C07289=1044.179,214.469,399.618,171.280,39.054,157.394
C07290=1044.186,214.718,399.591,171.283,39.057,157.395
C07291=1044.193,214.967,399.564,171.286,39.059,157.395
C07292=1044.198,215.215,399.538,171.287,39.062,157.396
C07293=1044.206,215.464,399.511,171.290,39.064,157.396
C07294=1044.212,215.712,399.483,171.291,39.067,157.397
C07295=1044.219,215.960,399.457,171.294,39.069,157.397
C07296=1044.225,216.209,399.430,171.296,39.072,157.398
C07297=1044.232,216.458,399.403,171.298,39.074,157.399
C07298=1044.238,216.706,399.377,171.300,39.077,157.399
C07299=1044.245,216.955,399.350,171.303,39.079,157.400
C07300=1044.251,217.202,399.323,171.306,39.082,157.400
C07301=1044.258,217.451,399.296,171.307,39.084,157.401
C07302=1044.265,217.700,399.268,171.310,39.087,157.402
C07303=1044.272,217.948,399.242,171.312,39.089,157.402
C07304=1044.277,218.197,399.215,171.314,39.091,157.403
C07305=1044.285,218.445,399.188,171.316,39.094,157.403
C07306=1044.291,218.694,399.161,171.319,39.096,157.404
C07307=1044.298,218.941,399.134,171.320,39.099,157.404
C07308=1044.304,219.190,399.107,171.323,39.101,157.405
C07309=1044.311,219.439,399.079,171.325,39.103,157.406
C07310=1044.318,219.688,399.053,171.328,39.106,157.406
C07311=1044.324,219.936,399.026,171.329,39.109,157.407
C07312=1044.331,220.184,398.999,171.332,39.111,157.407
C07313=1044.338,220.475,398.967,171.335,39.114,157.408
C07314=1044.346,220.766,398.935,171.337,39.117,157.409
C07315=1044.353,221.056,398.903,171.340,39.120,157.409
C07316=1044.362,221.347,398.871,171.343,39.123,157.410
C07317=1044.367,221.596,398.845,171.345,39.125,157.411
C07318=1044.374,221.844,398.817,171.347,39.128,157.411
C07319=1044.381,222.093,398.790,171.349,39.130,157.412
C07320=1044.387,222.341,398.763,171.352,39.133,157.412
C07321=1044.394,222.589,398.735,171.354,39.135,157.413
C07322=1044.400,222.838,398.708,171.356,39.138,157.414
C07323=1044.407,223.087,398.681,171.358,39.140,157.414
C07324=1044.413,223.334,398.653,171.361,39.142,157.415
C07325=1044.420,223.583,398.626,171.364,39.145,157.415
C07326=1044.427,223.831,398.599,171.365,39.148,157.416
C07327=1044.434,224.080,398.571,171.368,39.150,157.417
C07328=1044.439,224.328,398.545,171.370,39.152,157.417
C07329=1044.446,224.577,398.517,171.373,39.155,157.418
C07330=1044.453,224.825,398.489,171.374,39.158,157.418
C07331=1044.459,225.074,398.461,171.377,39.160,157.419
C07332=1044.466,225.323,398.434,171.379,39.162,157.420
C07333=1044.472,225.570,398.407,171.382,39.164,157.420
C07334=1044.479,225.819,398.380,171.385,39.167,157.421
C07335=1044.486,226.067,398.352,171.386,39.170,157.421
C07336=1044.492,226.316,398.325,171.389,39.172,157.422
C07337=1044.499,226.564,398.297,171.391,39.174,157.422
C07338=1044.506,226.813,398.270,171.394,39.177,157.423
C07339=1044.512,227.061,398.242,171.396,39.179,157.424
C07340=1044.519,227.309,398.215,171.398,39.182,157.424
C07341=1044.525,227.558,398.188,171.400,39.184,157.425
C07342=1044.532,227.807,398.160,171.403,39.186,157.425
C07343=1044.539,228.055,398.133,171.405,39.189,157.426
C07344=1044.546,228.303,398.105,171.408,39.192,157.427
C07345=1044.552,228.552,398.077,171.410,39.194,157.427
C07346=1044.559,228.800,398.050,171.412,39.196,157.428
C07347=1044.565,229.048,398.022,171.415,39.199,157.428
C07348=1044.572,229.296,397.994,171.417,39.201,157.429
C07349=1044.578,229.545,397.966,171.420,39.204,157.429
C07350=1044.584,229.793,397.938,171.421,39.206,157.430
C07351=1044.591,230.042,397.911,171.424,39.208,157.431
C07352=1044.598,230.290,397.883,171.427,39.211,157.431
C07353=1044.604,230.539,397.855,171.429,39.214,157.432
C07354=1044.611,230.786,397.828,171.432,39.216,157.432
C07355=1044.617,231.035,397.800,171.434,39.218,157.433
C07356=1044.624,231.283,397.772,171.436,39.221,157.434
C07357=1044.631,231.532,397.745,171.438,39.223,157.434
C07358=1044.637,231.781,397.716,171.441,39.226,157.435
C07359=1044.643,232.029,397.689,171.443,39.228,157.435
C07360=1044.650,232.277,397.661,171.446,39.231,157.436
C07361=1044.657,232.526,397.633,171.449,39.233,157.437
C07362=1044.663,232.774,397.605,171.451,39.236,157.437
C07363=1044.669,233.023,397.577,171.453,39.238,157.438
C07364=1044.675,233.271,397.550,171.455,39.241,157.438
C07365=1044.682,233.519,397.521,171.458,39.243,157.439
C07366=1044.689,233.767,397.494,171.461,39.246,157.440
C07367=1044.695,234.016,397.465,171.463,39.248,157.440
C07368=1044.702,234.264,397.438,171.466,39.251,157.441
C07369=1044.709,234.547,397.405,171.468,39.253,157.441
C07370=1044.717,234.831,397.373,171.471,39.256,157.442
C07371=1044.724,235.114,397.342,171.474,39.259,157.443
C07372=1044.731,235.397,397.309,171.476,39.262,157.444
C07373=1044.738,235.646,397.282,171.479,39.264,157.444
C07374=1044.745,235.894,397.254,171.481,39.267,157.445
C07375=1044.751,236.142,397.225,171.484,39.269,157.445
C07376=1044.758,236.391,397.197,171.487,39.272,157.446
C07377=1044.764,236.639,397.169,171.489,39.274,157.447
C07378=1044.771,236.887,397.142,171.492,39.276,157.447
C07379=1044.777,237.136,397.113,171.494,39.279,157.448
C07380=1044.784,237.384,397.085,171.497,39.282,157.448
C07381=1044.790,237.632,397.057,171.498,39.284,157.449
C07382=1044.797,237.881,397.028,171.501,39.286,157.449
C07383=1044.803,238.129,397.000,171.504,39.289,157.450
C07384=1044.810,238.377,396.972,171.506,39.291,157.451
C07385=1044.816,238.626,396.944,171.509,39.294,157.451
C07386=1044.823,238.874,396.916,171.511,39.296,157.452
C07387=1044.830,239.122,396.887,171.514,39.299,157.453
C07388=1044.837,239.371,396.859,171.516,39.301,157.453
C07389=1044.844,239.619,396.830,171.519,39.303,157.454
C07390=1044.850,239.868,396.803,171.521,39.306,157.454
C07391=1044.856,240.116,396.774,171.524,39.309,157.455
C07392=1044.863,240.364,396.746,171.527,39.311,157.455
C07393=1044.870,240.613,396.718,171.529,39.313,157.456
C07394=1044.876,240.861,396.689,171.532,39.315,157.457
C07395=1044.883,241.109,396.661,171.534,39.318,157.457
C07396=1044.889,241.357,396.632,171.537,39.321,157.458
C07397=1044.896,241.606,396.605,171.540,39.323,157.458
C07398=1044.902,241.854,396.575,171.542,39.326,157.459
C07399=1044.909,242.102,396.547,171.545,39.328,157.460
C07400=1044.915,242.350,396.519,171.547,39.330,157.460
C07401=1044.922,242.599,396.489,171.550,39.333,157.461
C07402=1044.929,242.847,396.461,171.553,39.335,157.462
C07403=1044.935,243.096,396.433,171.554,39.338,157.462
C07404=1044.942,243.344,396.404,171.557,39.341,157.463
C07405=1044.948,243.592,396.376,171.559,39.343,157.463
C07406=1044.954,243.841,396.347,171.562,39.345,157.464
C07407=1044.961,244.088,396.318,171.564,39.348,157.465
C07408=1044.967,244.336,396.289,171.567,39.350,157.465
C07409=1044.974,244.585,396.262,171.570,39.353,157.466
C07410=1044.981,244.834,396.232,171.572,39.355,157.466
C07411=1044.987,245.082,396.203,171.575,39.358,157.467
C07412=1044.994,245.330,396.175,171.577,39.360,157.468
C07413=1045.000,245.578,396.146,171.580,39.363,157.468
C07414=1045.006,245.827,396.117,171.583,39.365,157.469
C07415=1045.012,246.075,396.088,171.585,39.368,157.470
C07416=1045.019,246.323,396.060,171.588,39.370,157.470
C07417=1045.026,246.571,396.031,171.590,39.373,157.471
C07418=1045.032,246.820,396.002,171.593,39.375,157.471
C07419=1045.038,247.068,395.973,171.596,39.378,157.472
C07420=1045.045,247.316,395.944,171.598,39.381,157.473
C07421=1045.051,247.565,395.915,171.601,39.383,157.473
C07422=1045.057,247.813,395.886,171.603,39.386,157.474
C07423=1045.064,248.060,395.857,171.606,39.388,157.474
C07424=1045.070,248.309,395.828,171.610,39.390,157.475
C07425=1045.077,248.587,395.796,171.612,39.393,157.476
C07426=1045.085,248.864,395.764,171.615,39.396,157.476
C07427=1045.092,249.141,395.731,171.618,39.399,157.477
C07428=1045.099,249.419,395.698,171.621,39.402,157.478
C07429=1045.106,249.667,395.670,171.624,39.405,157.479
C07430=1045.112,249.915,395.641,171.627,39.407,157.479
C07431=1045.119,250.164,395.611,171.629,39.409,157.480
C07432=1045.125,250.412,395.582,171.632,39.412,157.480
C07433=1045.131,250.660,395.553,171.634,39.414,157.481
C07434=1045.137,250.908,395.524,171.637,39.417,157.482
C07435=1045.144,251.157,395.495,171.640,39.419,157.482
C07436=1045.151,251.405,395.466,171.642,39.422,157.483
C07437=1045.157,251.653,395.437,171.645,39.424,157.484
C07438=1045.164,251.900,395.408,171.647,39.427,157.484
C07439=1045.171,252.149,395.378,171.650,39.430,157.485
C07440=1045.177,252.397,395.349,171.654,39.432,157.485
C07441=1045.183,252.646,395.320,171.656,39.434,157.486
C07442=1045.190,252.894,395.291,171.659,39.437,157.487
C07443=1045.197,253.143,395.262,171.661,39.439,157.487
C07444=1045.203,253.391,395.233,171.664,39.442,157.488
C07445=1045.209,253.639,395.204,171.667,39.444,157.488
C07446=1045.216,253.887,395.174,171.669,39.447,157.489
C07447=1045.222,254.135,395.145,171.672,39.449,157.490
C07448=1045.229,254.383,395.115,171.674,39.452,157.490
C07449=1045.236,254.632,395.087,171.678,39.454,157.491
C07450=1045.243,254.879,395.057,171.681,39.457,157.492
C07451=1045.249,255.127,395.028,171.683,39.459,157.492
C07452=1045.256,255.376,394.998,171.686,39.462,157.493
C07453=1045.262,255.624,394.969,171.688,39.464,157.493
C07454=1045.269,255.872,394.940,171.691,39.466,157.494
C07455=1045.276,256.121,394.910,171.694,39.469,157.495
C07456=1045.282,256.369,394.881,171.697,39.471,157.495
C07457=1045.289,256.618,394.852,171.700,39.474,157.496
C07458=1045.295,256.865,394.822,171.702,39.477,157.497
C07459=1045.302,257.113,394.793,171.705,39.479,157.497
C07460=1045.308,257.362,394.764,171.708,39.482,157.498
C07461=1045.315,257.610,394.734,171.710,39.484,157.498
C07462=1045.322,257.859,394.704,171.714,39.486,157.499
C07463=1045.329,258.106,394.675,171.717,39.489,157.500
C07464=1045.335,258.354,394.646,171.719,39.491,157.500
C07465=1045.342,258.603,394.617,171.722,39.494,157.501
C07466=1045.349,258.850,394.587,171.724,39.496,157.502
C07467=1045.356,259.099,394.558,171.728,39.498,157.502
C07468=1045.362,259.347,394.528,171.731,39.501,157.503
C07469=1045.369,259.595,394.499,171.733,39.504,157.503
C07470=1045.376,259.843,394.469,171.736,39.506,157.504
C07471=1045.382,260.092,394.439,171.738,39.509,157.505
C07472=1045.389,260.339,394.410,171.742,39.511,157.505
C07473=1045.396,260.588,394.380,171.745,39.513,157.506
C07474=1045.402,260.836,394.350,171.747,39.516,157.507
C07475=1045.409,261.084,394.321,171.750,39.518,157.507
C07476=1045.416,261.332,394.291,171.754,39.521,157.508
C07477=1045.423,261.581,394.262,171.756,39.523,157.508
C07478=1045.429,261.828,394.232,171.759,39.525,157.509
C07479=1045.436,262.077,394.203,171.761,39.528,157.510
C07480=1045.443,262.325,394.173,171.765,39.530,157.510
C07481=1045.450,262.600,394.140,171.768,39.533,157.511
C07482=1045.457,262.876,394.106,171.771,39.536,157.512
C07483=1045.465,263.153,394.074,171.774,39.539,157.513
C07484=1045.472,263.429,394.040,171.778,39.542,157.513
C07485=1045.479,263.677,394.010,171.780,39.545,157.514
C07486=1045.485,263.925,393.980,171.783,39.547,157.515
C07487=1045.492,264.173,393.950,171.786,39.550,157.515
C07488=1045.498,264.421,393.921,171.788,39.552,157.516
C07489=1045.505,264.670,393.890,171.792,39.555,157.517
C07490=1045.511,264.917,393.860,171.794,39.557,157.517
C07491=1045.518,265.165,393.830,171.797,39.560,157.518
C07492=1045.524,265.413,393.800,171.801,39.563,157.519
C07493=1045.531,265.662,393.770,171.803,39.565,157.519
C07494=1045.537,265.910,393.741,171.806,39.568,157.520
C07495=1045.544,266.158,393.710,171.809,39.570,157.520
C07496=1045.551,266.406,393.680,171.812,39.573,157.521
C07497=1045.558,266.654,393.650,171.815,39.575,157.522
C07498=1045.564,266.902,393.619,171.818,39.578,157.522
C07499=1045.571,267.150,393.589,171.820,39.580,157.523
C07500=1045.578,267.398,393.559,171.824,39.583,157.524
C07501=1045.584,267.647,393.529,171.827,39.585,157.524
C07502=1045.591,267.894,393.499,171.829,39.588,157.525
C07503=1045.597,268.143,393.468,171.833,39.591,157.526
C07504=1045.604,268.390,393.438,171.836,39.593,157.526
C07505=1045.610,268.639,393.408,171.838,39.596,157.527
C07506=1045.617,268.886,393.378,171.842,39.598,157.528
C07507=1045.623,269.135,393.347,171.845,39.601,157.528
C07508=1045.630,269.383,393.317,171.847,39.603,157.529
C07509=1045.636,269.631,393.287,171.851,39.606,157.530
C07510=1045.643,269.879,393.257,171.854,39.609,157.530
C07511=1045.650,270.127,393.226,171.856,39.611,157.531
C07512=1045.656,270.375,393.196,171.859,39.614,157.532
C07513=1045.663,270.624,393.165,171.863,39.616,157.532
C07514=1045.670,270.872,393.135,171.865,39.619,157.533
C07515=1045.676,271.119,393.104,171.869,39.621,157.534
C07516=1045.683,271.367,393.074,171.871,39.624,157.534
C07517=1045.689,271.616,393.043,171.874,39.626,157.535
C07518=1045.696,271.863,393.014,171.878,39.629,157.536
C07519=1045.702,272.112,392.983,171.880,39.631,157.536
C07520=1045.709,272.360,392.952,171.883,39.634,157.537
C07521=1045.716,272.607,392.922,171.887,39.637,157.538
C07522=1045.722,272.856,392.891,171.889,39.639,157.538
C07523=1045.729,273.104,392.860,171.892,39.642,157.539
C07524=1045.735,273.351,392.830,171.896,39.645,157.540
C07525=1045.742,273.600,392.799,171.898,39.647,157.540
C07526=1045.748,273.848,392.768,171.901,39.650,157.541
C07527=1045.755,274.095,392.738,171.905,39.653,157.542
C07528=1045.762,274.344,392.707,171.907,39.655,157.542
C07529=1045.768,274.592,392.677,171.911,39.658,157.543
C07530=1045.775,274.840,392.646,171.914,39.660,157.544
C07531=1045.781,275.087,392.615,171.916,39.663,157.544
C07532=1045.788,275.336,392.585,171.920,39.665,157.545
C07533=1045.794,275.584,392.553,171.923,39.668,157.546
C07534=1045.802,275.832,392.523,171.927,39.671,157.547
C07535=1045.808,276.079,392.492,171.929,39.673,157.547
C07536=1045.814,276.328,392.461,171.932,39.676,157.548
C07537=1045.825,276.739,392.410,171.937,39.681,157.549
C07538=1045.832,276.982,392.380,171.941,39.683,157.550
C07539=1045.838,277.225,392.350,171.943,39.686,157.550
C07540=1045.845,277.468,392.319,171.946,39.688,157.551
C07541=1045.851,277.711,392.289,171.950,39.691,157.552
C07542=1045.858,277.954,392.258,171.952,39.693,157.552
C07543=1045.865,278.198,392.228,171.956,39.696,157.553
C07544=1045.871,278.441,392.198,171.959,39.698,157.554
C07545=1045.877,278.690,392.167,171.961,39.701,157.554
C07546=1045.884,278.937,392.136,171.965,39.704,157.555
C07547=1045.891,279.185,392.105,171.968,39.707,157.556
C07548=1045.897,279.433,392.074,171.971,39.709,157.557
C07549=1045.904,279.681,392.043,171.974,39.712,157.557
C07550=1045.911,279.929,392.011,171.978,39.714,157.558
C07551=1045.917,280.177,391.981,171.980,39.717,157.559
C07552=1045.923,280.425,391.950,171.984,39.720,157.559
C07553=1045.930,280.672,391.918,171.987,39.723,157.560
C07554=1045.937,280.920,391.887,171.990,39.726,157.561
C07555=1045.943,281.169,391.856,171.993,39.728,157.561
C07556=1045.950,281.417,391.825,171.996,39.731,157.562
C07557=1045.957,281.665,391.793,172.000,39.733,157.563
C07558=1045.963,281.912,391.762,172.002,39.736,157.564
C07559=1045.969,282.160,391.730,172.006,39.739,157.564
C07560=1045.976,282.408,391.699,172.009,39.742,157.565
C07561=1045.982,282.657,391.668,172.013,39.744,157.566
C07562=1045.989,282.904,391.637,172.015,39.747,157.566
C07563=1045.995,283.152,391.605,172.019,39.749,157.567
C07564=1046.002,283.400,391.574,172.022,39.752,157.568
C07565=1046.009,283.648,391.542,172.025,39.755,157.568
C07566=1046.016,283.896,391.511,172.028,39.758,157.569
C07567=1046.022,284.144,391.479,172.032,39.760,157.570
C07568=1046.029,284.392,391.448,172.035,39.763,157.571
C07569=1046.036,284.640,391.416,172.038,39.766,157.571
C07570=1046.043,284.888,391.385,172.041,39.769,157.572
C07571=1046.049,285.136,391.354,172.045,39.772,157.573
C07572=1046.056,285.383,391.322,172.047,39.774,157.573
C07573=1046.063,285.631,391.291,172.051,39.776,157.574
C07574=1046.069,285.879,391.259,172.055,39.779,157.575
C07575=1046.076,286.127,391.228,172.058,39.782,157.576
C07576=1046.083,286.375,391.196,172.061,39.785,157.576
C07577=1046.090,286.623,391.165,172.064,39.788,157.577
C07578=1046.096,286.871,391.134,172.068,39.790,157.578
C07579=1046.103,287.119,391.102,172.070,39.793,157.579
C07580=1046.110,287.367,391.071,172.074,39.796,157.579
C07581=1046.116,287.615,391.039,172.078,39.799,157.580
C07582=1046.123,287.862,391.007,172.081,39.801,157.581
C07583=1046.130,288.110,390.975,172.084,39.804,157.581
C07584=1046.136,288.358,390.944,172.087,39.807,157.582
C07585=1046.142,288.606,390.912,172.091,39.810,157.583
C07586=1046.149,288.853,390.880,172.094,39.812,157.584
C07587=1046.156,289.101,390.848,172.097,39.815,157.584
C07588=1046.163,289.349,390.817,172.101,39.818,157.585
C07589=1046.169,289.598,390.785,172.104,39.821,157.586
C07590=1046.176,289.845,390.752,172.108,39.823,157.587
C07591=1046.182,290.093,390.721,172.110,39.826,157.587
C07592=1046.189,290.341,390.690,172.114,39.829,157.588
C07593=1046.197,290.633,390.652,172.118,39.832,157.589
C07594=1046.205,290.924,390.613,172.122,39.835,157.590
C07595=1046.212,291.216,390.576,172.126,39.839,157.591
C07596=1046.220,291.509,390.538,172.130,39.842,157.592
C07597=1046.227,291.757,390.506,172.133,39.845,157.592
C07598=1046.234,292.004,390.474,172.136,39.848,157.593
C07599=1046.240,292.252,390.442,172.140,39.850,157.594
C07600=1046.247,292.500,390.410,172.144,39.853,157.595
C07601=1046.254,292.748,390.379,172.146,39.856,157.595
C07602=1046.260,292.995,390.346,172.150,39.859,157.596
C07603=1046.268,293.244,390.314,172.154,39.862,157.597
C07604=1046.275,293.491,390.282,172.157,39.865,157.598
C07605=1046.281,293.739,390.250,172.160,39.867,157.598
C07606=1046.288,293.987,390.218,172.164,39.870,157.599
C07607=1046.294,294.235,390.186,172.167,39.873,157.600
C07608=1046.301,294.482,390.154,172.171,39.876,157.601
C07609=1046.308,294.730,390.121,172.174,39.878,157.601
C07610=1046.314,294.978,390.089,172.177,39.882,157.602
C07611=1046.321,295.226,390.056,172.181,39.884,157.603
C07612=1046.328,295.473,390.024,172.185,39.887,157.604
C07613=1046.334,295.721,389.993,172.187,39.890,157.604
C07614=1046.341,295.969,389.960,172.191,39.893,157.605
C07615=1046.348,296.217,389.927,172.195,39.896,157.606
C07616=1046.354,296.465,389.894,172.198,39.899,157.607
C07617=1046.361,296.712,389.863,172.202,39.901,157.607
C07618=1046.367,296.960,389.830,172.206,39.905,157.608
C07619=1046.373,297.208,389.797,172.208,39.908,157.609
C07620=1046.380,297.456,389.764,172.212,39.910,157.610
C07621=1046.386,297.703,389.731,172.216,39.914,157.611
C07622=1046.393,297.951,389.699,172.219,39.916,157.611
C07623=1046.400,298.198,389.667,172.223,39.920,157.612
C07624=1046.407,298.447,389.633,172.226,39.922,157.613
C07625=1046.413,298.695,389.601,172.229,39.925,157.614
C07626=1046.420,298.942,389.569,172.233,39.928,157.615
C07627=1046.426,299.190,389.537,172.237,39.931,157.615
C07628=1046.433,299.438,389.503,172.241,39.934,157.616
C07629=1046.439,299.686,389.471,172.243,39.937,157.617
C07630=1046.445,299.933,389.438,172.247,39.940,157.618
C07631=1046.452,300.180,389.406,172.251,39.943,157.619
C07632=1046.459,300.429,389.373,172.254,39.946,157.619
C07633=1046.466,300.676,389.339,172.258,39.949,157.620
C07634=1046.472,300.923,389.306,172.261,39.952,157.621
C07635=1046.479,301.172,389.273,172.265,39.955,157.622
C07636=1046.485,301.419,389.241,172.268,39.958,157.623
C07637=1046.492,301.667,389.208,172.272,39.961,157.623
C07638=1046.499,301.915,389.175,172.276,39.964,157.624
C07639=1046.506,302.162,389.143,172.279,39.967,157.625
C07640=1046.512,302.410,389.110,172.282,39.970,157.626
C07641=1046.519,302.658,389.077,172.286,39.973,157.627
C07642=1046.525,302.905,389.043,172.290,39.975,157.627
C07643=1046.532,303.153,389.011,172.294,39.979,157.628
C07644=1046.539,303.401,388.978,172.298,39.981,157.629
C07645=1046.546,303.648,388.945,172.300,39.985,157.630
C07646=1046.553,303.896,388.912,172.304,39.987,157.631
C07647=1046.559,304.144,388.879,172.308,39.991,157.632
C07648=1046.565,304.391,388.846,172.312,39.993,157.632
C07649=1046.575,304.699,388.805,172.316,39.997,157.633
C07650=1046.582,305.008,388.764,172.321,40.001,157.634
C07651=1046.591,305.316,388.723,172.325,40.005,157.635
C07652=1046.600,305.624,388.681,172.330,40.009,157.636
C07653=1046.606,305.872,388.648,172.334,40.011,157.637
C07654=1046.613,306.120,388.615,172.338,40.015,157.638
C07655=1046.620,306.367,388.582,172.341,40.017,157.639
C07656=1046.627,306.615,388.549,172.344,40.021,157.640
C07657=1046.634,306.862,388.516,172.348,40.023,157.640
C07658=1046.641,307.111,388.482,172.352,40.027,157.641
C07659=1046.647,307.358,388.450,172.356,40.029,157.642
C07660=1046.654,307.606,388.416,172.360,40.033,157.643
C07661=1046.661,307.853,388.383,172.364,40.035,157.644
C07662=1046.668,308.101,388.349,172.368,40.039,157.645
C07663=1046.675,308.348,388.317,172.370,40.042,157.646
C07664=1046.682,308.596,388.283,172.374,40.045,157.646
C07665=1046.689,308.844,388.250,172.378,40.048,157.647
C07666=1046.696,309.091,388.217,172.382,40.051,157.648
C07667=1046.703,309.339,388.183,172.386,40.054,157.649
C07668=1046.709,309.587,388.150,172.390,40.057,157.650
C07669=1046.716,309.834,388.116,172.393,40.060,157.650
C07670=1046.723,310.082,388.083,172.397,40.063,157.651
C07671=1046.730,310.330,388.050,172.401,40.066,157.652
C07672=1046.737,310.577,388.016,172.405,40.069,157.653
C07673=1046.744,310.826,387.983,172.409,40.072,157.654
C07674=1046.751,311.072,387.950,172.412,40.075,157.655
C07675=1046.758,311.320,387.916,172.416,40.078,157.656
C07676=1046.766,311.568,387.882,172.420,40.082,157.656
C07677=1046.772,311.815,387.850,172.423,40.084,157.657
C07678=1046.779,312.063,387.816,172.427,40.087,157.658
C07679=1046.786,312.310,387.782,172.431,40.091,157.659
C07680=1046.794,312.558,387.748,172.435,40.093,157.660
C07681=1046.800,312.806,387.715,172.439,40.097,157.661
C07682=1046.806,313.054,387.681,172.443,40.100,157.662
C07683=1046.813,313.301,387.647,172.447,40.103,157.662
C07684=1046.819,313.549,387.613,172.451,40.106,157.663
C07685=1046.827,313.796,387.579,172.455,40.110,157.664
C07686=1046.834,314.044,387.546,172.459,40.113,157.665
C07687=1046.840,314.291,387.511,172.462,40.116,157.666
C07688=1046.847,314.539,387.478,172.466,40.119,157.667
C07689=1046.854,314.786,387.442,172.470,40.123,157.668
C07690=1046.860,315.033,387.409,172.474,40.126,157.669
C07691=1046.867,315.281,387.375,172.477,40.129,157.670
C07692=1046.874,315.529,387.341,172.481,40.133,157.670
C07693=1046.880,315.776,387.307,172.485,40.136,157.671
C07694=1046.887,316.024,387.273,172.489,40.139,157.672
C07695=1046.893,316.272,387.238,172.493,40.142,157.673
C07696=1046.901,316.520,387.205,172.497,40.146,157.674
C07697=1046.907,316.766,387.170,172.501,40.149,157.675
C07698=1046.914,317.014,387.136,172.505,40.152,157.676
C07699=1046.920,317.262,387.102,172.509,40.155,157.677
C07700=1046.928,317.510,387.068,172.513,40.159,157.678
C07701=1046.934,317.758,387.033,172.516,40.162,157.679
C07702=1046.941,318.004,386.999,172.520,40.165,157.679
C07703=1046.947,318.252,386.965,172.524,40.168,157.680
C07704=1046.955,318.500,386.931,172.528,40.172,157.681
C07705=1046.963,318.812,386.887,172.534,40.176,157.682
C07706=1046.971,319.125,386.844,172.539,40.180,157.684
C07707=1046.980,319.438,386.800,172.544,40.184,157.685
C07708=1046.989,319.751,386.757,172.549,40.188,157.686
C07709=1046.996,319.999,386.723,172.553,40.191,157.687
C07710=1047.003,320.246,386.688,172.557,40.195,157.688
C07711=1047.010,320.494,386.654,172.561,40.198,157.689
C07712=1047.016,320.740,386.619,172.565,40.202,157.690
C07713=1047.023,320.988,386.585,172.569,40.205,157.691
C07714=1047.030,321.235,386.551,172.573,40.208,157.691
C07715=1047.037,321.483,386.516,172.577,40.212,157.692
C07716=1047.044,321.730,386.481,172.581,40.215,157.693
C07717=1047.051,321.978,386.447,172.585,40.218,157.694
C07718=1047.058,322.226,386.412,172.589,40.222,157.695
C07719=1047.065,322.473,386.378,172.593,40.225,157.696
C07720=1047.072,322.721,386.343,172.598,40.228,157.697
C07721=1047.079,322.968,386.309,172.602,40.231,157.698
C07722=1047.086,323.216,386.274,172.606,40.235,157.699
C07723=1047.092,323.463,386.239,172.610,40.238,157.700
C07724=1047.100,323.711,386.205,172.614,40.242,157.701
C07725=1047.106,323.958,386.170,172.618,40.245,157.702
C07726=1047.114,324.206,386.135,172.622,40.248,157.703
C07727=1047.121,324.454,386.101,172.626,40.252,157.704
C07728=1047.128,324.701,386.066,172.631,40.255,157.705
C07729=1047.135,324.948,386.031,172.635,40.258,157.705
C07730=1047.142,325.196,385.997,172.639,40.262,157.707
C07731=1047.149,325.443,385.962,172.643,40.265,157.707
C07732=1047.156,325.691,385.927,172.647,40.269,157.708
C07733=1047.163,325.938,385.892,172.651,40.272,157.709
C07734=1047.170,326.185,385.857,172.656,40.275,157.710
C07735=1047.177,326.434,385.822,172.660,40.279,157.711
C07736=1047.185,326.681,385.788,172.664,40.283,157.712
C07737=1047.192,326.928,385.753,172.668,40.286,157.713
C07738=1047.198,327.175,385.718,172.672,40.289,157.714
C07739=1047.206,327.422,385.683,172.677,40.293,157.715
C07740=1047.213,327.671,385.648,172.681,40.296,157.716
C07741=1047.220,327.918,385.612,172.685,40.300,157.717
C07742=1047.227,328.165,385.578,172.689,40.303,157.718
C07743=1047.234,328.412,385.543,172.693,40.306,157.719
C07744=1047.242,328.660,385.508,172.698,40.310,157.720
C07745=1047.249,328.907,385.473,172.702,40.313,157.721
C07746=1047.256,329.155,385.438,172.706,40.317,157.722
C07747=1047.263,329.402,385.403,172.710,40.320,157.723
C07748=1047.271,329.650,385.368,172.715,40.324,157.724
C07749=1047.277,329.897,385.332,172.719,40.327,157.725
C07750=1047.284,330.145,385.297,172.723,40.331,157.726
C07751=1047.291,330.392,385.262,172.727,40.335,157.727
C07752=1047.299,330.639,385.226,172.732,40.338,157.728
C07753=1047.305,330.887,385.191,172.736,40.341,157.729
C07754=1047.312,331.134,385.156,172.740,40.345,157.730
C07755=1047.319,331.382,385.121,172.744,40.349,157.731
C07756=1047.327,331.629,385.084,172.748,40.352,157.732
C07757=1047.333,331.876,385.049,172.753,40.356,157.733
C07758=1047.339,332.124,385.013,172.758,40.360,157.734
C07759=1047.347,332.372,384.977,172.762,40.363,157.735
C07760=1047.354,332.619,384.942,172.767,40.367,157.736
C07761=1047.362,332.926,384.898,172.772,40.371,157.737
C07762=1047.371,333.235,384.854,172.777,40.376,157.739
C07763=1047.381,333.542,384.809,172.783,40.381,157.740
C07764=1047.389,333.850,384.765,172.788,40.385,157.741
C07765=1047.396,334.098,384.730,172.792,40.389,157.742
C07766=1047.403,334.345,384.694,172.797,40.392,157.743
C07767=1047.410,334.592,384.659,172.802,40.396,157.744
C07768=1047.418,334.839,384.622,172.805,40.399,157.745
C07769=1047.425,335.087,384.587,172.811,40.403,157.746
C07770=1047.432,335.334,384.551,172.815,40.407,157.747
C07771=1047.439,335.581,384.515,172.819,40.411,157.748
C07772=1047.447,335.829,384.480,172.824,40.414,157.750
C07773=1047.454,336.076,384.444,172.828,40.418,157.751
C07774=1047.460,336.323,384.407,172.832,40.422,157.752
C07775=1047.468,336.571,384.372,172.837,40.425,157.753
C07776=1047.475,336.818,384.336,172.842,40.429,157.754
C07777=1047.482,337.065,384.299,172.846,40.433,157.755
C07778=1047.488,337.313,384.264,172.851,40.437,157.756
C07779=1047.496,337.560,384.228,172.855,40.440,157.757
C07780=1047.502,337.807,384.191,172.859,40.444,157.758
C07781=1047.510,338.055,384.155,172.864,40.448,157.759
C07782=1047.517,338.301,384.119,172.868,40.452,157.760
C07783=1047.524,338.549,384.083,172.873,40.456,157.761
C07784=1047.531,338.797,384.047,172.878,40.460,157.763
C07785=1047.538,339.044,384.011,172.882,40.463,157.764
C07786=1047.546,339.291,383.975,172.887,40.467,157.765
C07787=1047.552,339.539,383.939,172.891,40.471,157.766
C07788=1047.560,339.785,383.903,172.896,40.475,157.767
C07789=1047.567,340.033,383.867,172.901,40.479,157.768
C07790=1047.574,340.280,383.830,172.905,40.483,157.769
C07791=1047.581,340.527,383.794,172.910,40.486,157.770
C07792=1047.589,340.775,383.758,172.914,40.490,157.771
C07793=1047.596,341.022,383.721,172.919,40.494,157.772
C07794=1047.603,341.269,383.685,172.924,40.498,157.773
C07795=1047.610,341.517,383.648,172.929,40.502,157.775
C07796=1047.617,341.764,383.612,172.933,40.505,157.776
C07797=1047.625,342.010,383.575,172.938,40.509,157.777
C07798=1047.632,342.258,383.539,172.942,40.513,157.778
C07799=1047.640,342.506,383.502,172.946,40.517,157.779
C07800=1047.646,342.753,383.466,172.952,40.521,157.780
C07801=1047.654,343.000,383.430,172.956,40.525,157.781
C07802=1047.661,343.247,383.392,172.961,40.529,157.782
C07803=1047.668,343.494,383.356,172.965,40.533,157.784
C07804=1047.675,343.742,383.319,172.970,40.537,157.785
C07805=1047.683,343.989,383.283,172.975,40.541,157.786
C07806=1047.689,344.236,383.246,172.980,40.545,157.787
C07807=1047.696,344.483,383.209,172.984,40.549,157.788
C07808=1047.704,344.730,383.172,172.989,40.553,157.789
C07809=1047.711,344.978,383.136,172.994,40.557,157.790
C07810=1047.718,345.224,383.099,172.999,40.561,157.792
C07811=1047.725,345.472,383.062,173.003,40.565,157.793
C07812=1047.733,345.719,383.025,173.009,40.569,157.794
C07813=1047.740,345.967,382.988,173.013,40.573,157.795
C07814=1047.747,346.213,382.951,173.018,40.577,157.796
C07815=1047.754,346.461,382.914,173.023,40.581,157.797
C07816=1047.762,346.708,382.878,173.027,40.585,157.799
C07817=1047.770,347.012,382.832,173.033,40.591,157.800
C07818=1047.780,347.316,382.786,173.040,40.595,157.802
C07819=1047.788,347.619,382.740,173.045,40.601,157.803
C07820=1047.797,347.923,382.696,173.052,40.605,157.804
C07821=1047.804,348.170,382.658,173.056,40.610,157.806
C07822=1047.812,348.417,382.621,173.061,40.614,157.807
C07823=1047.819,348.665,382.585,173.066,40.618,157.808
C07824=1047.826,348.912,382.547,173.071,40.622,157.809
C07825=1047.834,349.159,382.509,173.076,40.626,157.810
C07826=1047.842,349.406,382.473,173.081,40.630,157.812
C07827=1047.848,349.654,382.436,173.086,40.635,157.813
C07828=1047.856,349.901,382.398,173.090,40.638,157.814
C07829=1047.864,350.148,382.361,173.095,40.642,157.815
C07830=1047.871,350.395,382.324,173.101,40.647,157.816
C07831=1047.878,350.642,382.286,173.105,40.651,157.818
C07832=1047.885,350.889,382.249,173.110,40.655,157.819
C07833=1047.893,351.136,382.211,173.116,40.659,157.820
C07834=1047.900,351.383,382.174,173.120,40.664,157.821
C07835=1047.907,351.631,382.136,173.125,40.668,157.823
C07836=1047.914,351.878,382.099,173.131,40.672,157.824
C07837=1047.922,352.125,382.061,173.135,40.676,157.825
C07838=1047.929,352.372,382.024,173.140,40.681,157.826
C07839=1047.936,352.619,381.986,173.146,40.685,157.828
C07840=1047.944,352.865,381.948,173.150,40.690,157.829
C07841=1047.952,353.112,381.911,173.156,40.694,157.830
C07842=1047.959,353.360,381.873,173.161,40.698,157.831
C07843=1047.966,353.607,381.836,173.165,40.702,157.833
C07844=1047.973,353.854,381.798,173.171,40.706,157.834
C07845=1047.981,354.100,381.760,173.176,40.711,157.835
C07846=1047.988,354.348,381.722,173.182,40.715,157.837
C07847=1047.995,354.595,381.685,173.186,40.720,157.838
C07848=1048.003,354.842,381.647,173.191,40.724,157.839
C07849=1048.010,355.088,381.609,173.197,40.728,157.840
C07850=1048.018,355.336,381.571,173.202,40.733,157.842
C07851=1048.026,355.583,381.533,173.206,40.737,157.843
C07852=1048.033,355.830,381.495,173.212,40.741,157.844
C07853=1048.040,356.077,381.458,173.217,40.746,157.846
C07854=1048.048,356.323,381.420,173.223,40.750,157.847
C07855=1048.056,356.571,381.382,173.227,40.754,157.848
C07856=1048.063,356.818,381.344,173.233,40.759,157.849
C07857=1048.070,357.065,381.306,173.238,40.763,157.851
C07858=1048.078,357.311,381.268,173.243,40.768,157.852
C07859=1048.084,357.559,381.230,173.249,40.772,157.853
C07860=1048.093,357.806,381.191,173.253,40.777,157.855
C07861=1048.100,358.053,381.153,173.259,40.781,157.856
C07862=1048.107,358.300,381.115,173.264,40.786,157.857
C07863=1048.115,358.546,381.077,173.270,40.790,157.859
C07864=1048.123,358.793,381.038,173.275,40.795,157.860
C07865=1048.130,359.040,381.000,173.280,40.800,157.861
C07866=1048.137,359.287,380.962,173.285,40.804,157.863
C07867=1048.145,359.535,380.923,173.291,40.809,157.864
C07868=1048.153,359.781,380.885,173.296,40.813,157.865
C07869=1048.160,360.028,380.847,173.302,40.818,157.867
C07870=1048.168,360.275,380.808,173.307,40.822,157.868
C07871=1048.175,360.522,380.770,173.313,40.827,157.869
C07872=1048.183,360.769,380.732,173.317,40.831,157.871
C07873=1048.193,361.078,380.683,173.324,40.837,157.872
C07874=1048.201,361.387,380.635,173.331,40.843,157.874
C07875=1048.211,361.697,380.587,173.338,40.849,157.876
C07876=1048.221,362.007,380.538,173.345,40.855,157.878
C07877=1048.228,362.253,380.500,173.350,40.859,157.879
C07878=1048.236,362.500,380.461,173.356,40.864,157.880
C07879=1048.243,362.747,380.422,173.361,40.868,157.882
C07880=1048.251,362.994,380.384,173.367,40.873,157.883
C07881=1048.259,363.241,380.345,173.372,40.878,157.885
C07882=1048.266,363.488,380.307,173.377,40.883,157.886
C07883=1048.274,363.734,380.267,173.382,40.887,157.887
C07884=1048.281,363.981,380.228,173.388,40.892,157.889
C07885=1048.288,364.229,380.189,173.394,40.897,157.890
C07886=1048.296,364.475,380.151,173.399,40.902,157.892
C07887=1048.304,364.722,380.111,173.405,40.907,157.893
C07888=1048.311,364.969,380.073,173.410,40.912,157.895
C07889=1048.319,365.216,380.034,173.416,40.916,157.896
C07890=1048.327,365.462,379.995,173.421,40.921,157.897
C07891=1048.334,365.709,379.955,173.427,40.926,157.899
C07892=1048.342,365.955,379.916,173.433,40.931,157.900
C07893=1048.349,366.203,379.877,173.438,40.936,157.902
C07894=1048.358,366.449,379.838,173.444,40.940,157.903
C07895=1048.365,366.696,379.799,173.450,40.946,157.905
C07896=1048.373,366.943,379.760,173.455,40.950,157.906
C07897=1048.380,367.190,379.721,173.461,40.955,157.907
C07898=1048.388,367.437,379.681,173.466,40.960,157.909
C07899=1048.396,367.683,379.642,173.472,40.965,157.910
C07900=1048.403,367.930,379.603,173.478,40.970,157.912
C07901=1048.411,368.177,379.564,173.483,40.975,157.913
C07902=1048.419,368.424,379.524,173.489,40.980,157.915
C07903=1048.427,368.670,379.485,173.496,40.985,157.916
C07904=1048.434,368.917,379.445,173.501,40.989,157.918
C07905=1048.442,369.164,379.406,173.507,40.995,157.919
C07906=1048.450,369.410,379.366,173.513,41.000,157.921
C07907=1048.457,369.657,379.327,173.518,41.005,157.922
C07908=1048.466,369.904,379.288,173.524,41.010,157.924
C07909=1048.473,370.151,379.248,173.530,41.014,157.925
C07910=1048.481,370.398,379.208,173.535,41.020,157.927
C07911=1048.489,370.644,379.169,173.541,41.025,157.929
C07912=1048.497,370.890,379.129,173.548,41.029,157.930
C07913=1048.505,371.137,379.090,173.554,41.035,157.932
C07914=1048.513,371.384,379.050,173.559,41.040,157.933
C07915=1048.521,371.631,379.010,173.565,41.045,157.935
C07916=1048.528,371.878,378.970,173.571,41.050,157.936
C07917=1048.535,372.124,378.931,173.576,41.055,157.938
C07918=1048.543,372.371,378.891,173.583,41.060,157.939
C07919=1048.551,372.618,378.851,173.589,41.065,157.941
C07920=1048.560,372.864,378.811,173.595,41.071,157.942
C07921=1048.567,373.111,378.771,173.600,41.076,157.944
C07922=1048.575,373.358,378.731,173.606,41.081,157.946
C07923=1048.582,373.604,378.691,173.612,41.086,157.947
C07924=1048.590,373.850,378.651,173.619,41.091,157.949
C07925=1048.598,374.097,378.611,173.625,41.097,157.950
C07926=1048.606,374.344,378.571,173.630,41.102,157.952
C07927=1048.614,374.590,378.530,173.636,41.108,157.954
C07928=1048.621,374.837,378.490,173.643,41.113,157.955
C07929=1048.632,375.165,378.436,173.650,41.120,157.957
C07930=1048.643,375.494,378.383,173.659,41.127,157.959
C07931=1048.654,375.823,378.330,173.667,41.134,157.962
C07932=1048.664,376.151,378.276,173.675,41.141,157.964
C07933=1048.671,376.398,378.236,173.682,41.147,157.965
C07934=1048.680,376.645,378.195,173.687,41.152,157.967
C07935=1048.688,376.891,378.155,173.693,41.157,157.969
C07936=1048.696,377.138,378.115,173.700,41.163,157.970
C07937=1048.704,377.384,378.074,173.706,41.168,157.972
C07938=1048.712,377.630,378.033,173.712,41.173,157.973
C07939=1048.720,377.877,377.993,173.719,41.179,157.975
C07940=1048.728,378.124,377.953,173.725,41.184,157.977
C07941=1048.736,378.370,377.912,173.731,41.190,157.979
C07942=1048.744,378.616,377.871,173.737,41.195,157.980
C07943=1048.752,378.863,377.830,173.743,41.200,157.982
C07944=1048.760,379.110,377.791,173.749,41.206,157.984
C07945=1048.768,379.356,377.750,173.756,41.211,157.985
C07946=1048.776,379.603,377.709,173.762,41.217,157.987
C07947=1048.785,379.850,377.668,173.769,41.223,157.989
C07948=1048.793,380.096,377.628,173.775,41.228,157.990
C07949=1048.800,380.343,377.586,173.781,41.234,157.992
C07950=1048.808,380.589,377.546,173.788,41.239,157.994
C07951=1048.816,380.834,377.504,173.794,41.245,157.996
C07952=1048.825,381.081,377.463,173.801,41.251,157.997
C07953=1048.832,381.328,377.422,173.807,41.256,157.999
C07954=1048.840,381.574,377.382,173.814,41.262,158.001
C07955=1048.848,381.821,377.341,173.820,41.268,158.003
C07956=1048.857,382.067,377.299,173.826,41.273,158.004
C07957=1048.865,382.314,377.258,173.833,41.279,158.006
C07958=1048.873,382.560,377.217,173.839,41.285,158.008
C07959=1048.881,382.807,377.175,173.846,41.290,158.010
C07960=1048.889,383.053,377.134,173.852,41.296,158.011
C07961=1048.897,383.299,377.094,173.859,41.302,158.013
C07962=1048.906,383.546,377.052,173.865,41.307,158.015
C07963=1048.913,383.792,377.011,173.872,41.314,158.017
C07964=1048.921,384.038,376.970,173.878,41.319,158.018
C07965=1048.930,384.285,376.929,173.885,41.325,158.020
C07966=1048.938,384.531,376.887,173.891,41.331,158.022
C07967=1048.946,384.778,376.846,173.898,41.337,158.024
C07968=1048.954,385.024,376.804,173.905,41.342,158.026
C07969=1048.963,385.270,376.762,173.911,41.348,158.027
C07970=1048.971,385.516,376.721,173.918,41.354,158.029
C07971=1048.979,385.763,376.679,173.924,41.360,158.031
C07972=1048.987,386.009,376.638,173.932,41.366,158.033
C07973=1048.996,386.256,376.597,173.939,41.372,158.035
C07974=1049.004,386.502,376.555,173.945,41.378,158.037
C07975=1049.012,386.748,376.513,173.952,41.384,158.038
C07976=1049.021,386.994,376.472,173.958,41.390,158.040
C07977=1049.029,387.240,376.429,173.965,41.395,158.042
C07978=1049.038,387.487,376.388,173.972,41.402,158.044
C07979=1049.046,387.733,376.347,173.979,41.408,158.046
C07980=1049.054,387.980,376.305,173.986,41.413,158.048
C07981=1049.063,388.226,376.263,173.993,41.419,158.050
C07982=1049.071,388.472,376.221,174.000,41.426,158.052
C07983=1049.080,388.718,376.179,174.006,41.432,158.054
C07984=1049.089,388.965,376.138,174.013,41.437,158.055
C07985=1049.100,389.326,376.076,174.024,41.447,158.058
C07986=1049.113,389.687,376.013,174.034,41.456,158.061
C07987=1049.125,390.048,375.952,174.044,41.465,158.064
C07988=1049.137,390.410,375.890,174.055,41.474,158.067
C07989=1049.146,390.656,375.848,174.061,41.480,158.069
C07990=1049.154,390.902,375.805,174.068,41.486,158.071
C07991=1049.162,391.149,375.763,174.075,41.492,158.073
C07992=1049.171,391.395,375.721,174.083,41.499,158.075
C07993=1049.180,391.641,375.678,174.090,41.505,158.077
C07994=1049.188,391.886,375.636,174.096,41.511,158.078
C07995=1049.196,392.133,375.594,174.104,41.518,158.081
C07996=1049.205,392.379,375.551,174.111,41.524,158.083
C07997=1049.213,392.626,375.509,174.118,41.530,158.084
C07998=1049.222,392.872,375.466,174.126,41.537,158.087
C07999=1049.231,393.118,375.424,174.133,41.543,158.089
C08000=1049.239,393.364,375.381,174.139,41.550,158.091
C08001=1049.248,393.610,375.338,174.147,41.556,158.093
C08002=1049.255,393.856,375.295,174.154,41.562,158.095
C08003=1049.264,394.102,375.253,174.161,41.569,158.097
C08004=1049.273,394.348,375.210,174.169,41.575,158.099
C08005=1049.281,394.594,375.167,174.176,41.582,158.101
C08006=1049.290,394.840,375.124,174.184,41.588,158.103
C08007=1049.298,395.086,375.081,174.191,41.595,158.105
C08008=1049.307,395.332,375.038,174.198,41.601,158.107
C08009=1049.315,395.578,374.995,174.206,41.608,158.109
C08010=1049.325,395.825,374.952,174.213,41.614,158.111
C08011=1049.334,396.071,374.909,174.221,41.621,158.113
C08012=1049.342,396.317,374.866,174.228,41.627,158.115
C08013=1049.351,396.563,374.823,174.236,41.634,158.117
C08014=1049.359,396.809,374.780,174.243,41.641,158.120
C08015=1049.368,397.055,374.737,174.251,41.647,158.122
C08016=1049.376,397.301,374.694,174.258,41.654,158.124
C08017=1049.385,397.547,374.651,174.266,41.661,158.126
C08018=1049.394,397.793,374.607,174.273,41.668,158.128
C08019=1049.403,398.039,374.564,174.281,41.674,158.130
C08020=1049.411,398.285,374.521,174.288,41.681,158.132
C08021=1049.420,398.531,374.477,174.296,41.687,158.135
C08022=1049.428,398.777,374.434,174.303,41.695,158.137
C08023=1049.438,399.023,374.390,174.311,41.701,158.139
C08024=1049.446,399.269,374.347,174.319,41.708,158.141
C08025=1049.455,399.514,374.303,174.326,41.715,158.143
C08026=1049.464,399.762,374.259,174.334,41.722,158.146
C08027=1049.472,400.007,374.216,174.341,41.729,158.148
C08028=1049.481,400.253,374.173,174.349,41.736,158.150
C08029=1049.490,400.499,374.129,174.358,41.742,158.152
C08030=1049.499,400.745,374.086,174.365,41.749,158.154
C08031=1049.508,400.991,374.041,174.373,41.756,158.157
C08032=1049.517,401.237,373.998,174.380,41.763,158.159
C08033=1049.526,401.482,373.954,174.388,41.770,158.161
C08034=1049.534,401.729,373.910,174.397,41.777,158.163
C08035=1049.543,401.975,373.866,174.405,41.784,158.166
C08036=1049.552,402.221,373.822,174.412,41.791,158.168
C08037=1049.561,402.466,373.778,174.420,41.798,158.170
C08038=1049.570,402.713,373.734,174.428,41.806,158.173
C08039=1049.579,402.958,373.690,174.436,41.813,158.175
C08040=1049.588,403.204,373.646,174.444,41.820,158.177
C08041=1049.601,403.585,373.578,174.456,41.831,158.181
C08042=1049.616,403.965,373.509,174.469,41.842,158.184
C08043=1049.629,404.344,373.441,174.481,41.853,158.188
C08044=1049.643,404.724,373.372,174.494,41.864,158.192
C08045=1049.652,404.970,373.328,174.502,41.872,158.194
C08046=1049.661,405.217,373.283,174.510,41.879,158.196
C08047=1049.670,405.462,373.239,174.519,41.886,158.199
C08048=1049.679,405.708,373.194,174.527,41.894,158.201
C08049=1049.688,405.954,373.149,174.536,41.901,158.204
C08050=1049.697,406.199,373.105,174.544,41.908,158.206
C08051=1049.706,406.445,373.060,174.552,41.916,158.209
C08052=1049.715,406.691,373.016,174.560,41.923,158.211
C08053=1049.724,406.937,372.970,174.568,41.931,158.213
C08054=1049.733,407.183,372.926,174.577,41.938,158.216
C08055=1049.742,407.428,372.881,174.585,41.946,158.218
C08056=1049.752,407.674,372.836,174.594,41.953,158.221
C08057=1049.760,407.920,372.791,174.602,41.961,158.223
C08058=1049.770,408.166,372.747,174.611,41.968,158.226
C08059=1049.779,408.412,372.701,174.619,41.976,158.228
C08060=1049.789,408.657,372.656,174.628,41.983,158.231
C08061=1049.797,408.904,372.612,174.636,41.991,158.233
C08062=1049.806,409.149,372.566,174.645,41.998,158.236
C08063=1049.816,409.395,372.521,174.653,42.006,158.238
C08064=1049.825,409.641,372.476,174.662,42.014,158.241
C08065=1049.835,409.886,372.431,174.671,42.021,158.243
C08066=1049.844,410.132,372.386,174.679,42.029,158.246
C08067=1049.853,410.378,372.341,174.688,42.037,158.248
C08068=1049.862,410.623,372.296,174.697,42.045,158.251
C08069=1049.871,410.869,372.250,174.706,42.052,158.253
C08070=1049.881,411.114,372.205,174.715,42.060,158.256
C08071=1049.890,411.360,372.159,174.723,42.068,158.259
C08072=1049.901,411.606,372.114,174.732,42.076,158.261
C08073=1049.910,411.852,372.069,174.741,42.084,158.264
C08074=1049.919,412.097,372.022,174.750,42.091,158.266
C08075=1049.929,412.343,371.978,174.758,42.099,158.269
C08076=1049.938,412.589,371.932,174.768,42.107,158.272
C08077=1049.948,412.834,371.886,174.777,42.115,158.274
C08078=1049.957,413.080,371.841,174.786,42.123,158.277
C08079=1049.966,413.325,371.795,174.795,42.131,158.280
C08080=1049.976,413.572,371.749,174.804,42.139,158.282
C08081=1049.985,413.817,371.703,174.813,42.147,158.285
C08082=1049.995,414.062,371.657,174.822,42.155,158.288
C08083=1050.004,414.309,371.611,174.831,42.163,158.291
C08084=1050.013,414.554,371.565,174.841,42.171,158.293
C08085=1050.023,414.799,371.519,174.850,42.180,158.296
C08086=1050.033,415.045,371.472,174.858,42.188,158.299
C08087=1050.042,415.290,371.426,174.868,42.196,158.302
C08088=1050.053,415.536,371.380,174.877,42.204,158.304
C08089=1050.062,415.781,371.334,174.887,42.213,158.307
C08090=1050.071,416.026,371.288,174.896,42.221,158.310
C08091=1050.081,416.272,371.241,174.905,42.229,158.313
C08092=1050.090,416.517,371.195,174.915,42.237,158.316
C08093=1050.100,416.763,371.149,174.924,42.246,158.318
C08094=1050.110,417.009,371.102,174.934,42.254,158.321
C08095=1050.119,417.254,371.056,174.943,42.263,158.324
C08096=1050.129,417.500,371.010,174.953,42.271,158.327
C08097=1050.141,417.802,370.952,174.965,42.281,158.330
C08098=1050.153,418.105,370.894,174.976,42.292,158.334
C08099=1050.166,418.408,370.837,174.989,42.302,158.338
C08100=1050.177,418.710,370.780,175.000,42.313,158.341
C08101=1050.188,418.955,370.733,175.011,42.321,158.344
C08102=1050.197,419.201,370.686,175.020,42.330,158.347
C08103=1050.207,419.447,370.638,175.030,42.338,158.350
C08104=1050.217,419.692,370.592,175.040,42.347,158.353
C08105=1050.226,419.937,370.545,175.049,42.355,158.356
C08106=1050.237,420.182,370.498,175.060,42.364,158.359
C08107=1050.246,420.428,370.450,175.070,42.373,158.362
C08108=1050.256,420.674,370.403,175.079,42.381,158.365
C08109=1050.265,420.918,370.357,175.089,42.390,158.368
C08110=1050.276,421.164,370.309,175.100,42.399,158.371
C08111=1050.286,421.409,370.262,175.109,42.408,158.374
C08112=1050.295,421.655,370.214,175.119,42.417,158.377
C08113=1050.305,421.900,370.167,175.130,42.426,158.380
C08114=1050.316,422.145,370.120,175.140,42.435,158.383
C08115=1050.325,422.391,370.072,175.149,42.443,158.386
C08116=1050.335,422.636,370.025,175.160,42.452,158.389
C08117=1050.346,422.881,369.977,175.170,42.462,158.392
C08118=1050.356,423.126,369.930,175.181,42.470,158.395
C08119=1050.365,423.372,369.882,175.191,42.479,158.398
C08120=1050.376,423.617,369.835,175.202,42.488,158.402
C08121=1050.386,423.862,369.787,175.211,42.497,158.405
C08122=1050.396,424.107,369.740,175.222,42.506,158.408
C08123=1050.407,424.352,369.691,175.232,42.515,158.411
C08124=1050.417,424.598,369.643,175.243,42.525,158.414
C08125=1050.427,424.842,369.596,175.253,42.534,158.417
C08126=1050.437,425.088,369.548,175.264,42.543,158.421
C08127=1050.448,425.333,369.499,175.274,42.552,158.424
C08128=1050.457,425.579,369.452,175.285,42.561,158.427
C08129=1050.468,425.824,369.404,175.296,42.571,158.430
C08130=1050.478,426.069,369.355,175.306,42.580,158.434
C08131=1050.489,426.314,369.307,175.318,42.589,158.437
C08132=1050.498,426.559,369.258,175.329,42.599,158.440
C08133=1050.509,426.804,369.210,175.339,42.608,158.443
C08134=1050.519,427.049,369.162,175.350,42.618,158.447
C08135=1050.530,427.294,369.114,175.361,42.627,158.450
C08136=1050.540,427.539,369.065,175.372,42.637,158.453
C08137=1050.551,427.784,369.017,175.382,42.646,158.457
C08138=1050.560,428.029,368.968,175.394,42.656,158.460
C08139=1050.572,428.275,368.920,175.405,42.665,158.464
C08140=1050.582,428.519,368.871,175.416,42.674,158.467
C08141=1050.592,428.765,368.822,175.427,42.684,158.470
C08142=1050.602,429.009,368.774,175.439,42.694,158.474
C08143=1050.613,429.255,368.725,175.450,42.703,158.477
C08144=1050.624,429.500,368.676,175.461,42.713,158.481
C08145=1050.634,429.745,368.627,175.473,42.723,158.484
C08146=1050.645,429.990,368.578,175.484,42.732,158.487
C08147=1050.655,430.234,368.529,175.495,42.743,158.491
C08148=1050.666,430.479,368.480,175.507,42.752,158.494
C08149=1050.680,430.808,368.413,175.522,42.766,158.499
C08150=1050.694,431.137,368.347,175.537,42.779,158.504
C08151=1050.708,431.466,368.282,175.553,42.792,158.509
C08152=1050.722,431.794,368.215,175.569,42.806,158.514
C08153=1050.740,432.204,368.132,175.588,42.823,158.520
C08154=1050.758,432.614,368.049,175.608,42.839,158.526
C08155=1050.776,433.023,367.967,175.628,42.856,158.532
C08156=1050.794,433.433,367.883,175.648,42.874,158.538
C08157=1050.805,433.678,367.834,175.659,42.884,158.542
C08158=1050.816,433.922,367.784,175.671,42.894,158.545
C08159=1050.827,434.167,367.734,175.684,42.904,158.549
C08160=1050.838,434.412,367.684,175.695,42.914,158.553
C08161=1050.849,434.657,367.635,175.708,42.925,158.557
C08162=1050.860,434.901,367.584,175.720,42.935,158.560
C08163=1050.871,435.147,367.534,175.732,42.945,158.564
C08164=1050.883,435.391,367.484,175.745,42.956,158.568
C08165=1050.894,435.636,367.434,175.757,42.966,158.572
C08166=1050.905,435.880,367.384,175.769,42.977,158.576
C08167=1050.915,436.125,367.334,175.781,42.987,158.579
C08168=1050.927,436.370,367.284,175.794,42.998,158.583
C08169=1050.938,436.615,367.233,175.807,43.008,158.587
C08170=1050.949,436.859,367.183,175.819,43.019,158.591
C08171=1050.960,437.104,367.133,175.832,43.030,158.595
C08172=1050.971,437.349,367.082,175.844,43.040,158.599
C08173=1050.983,437.593,367.031,175.857,43.051,158.603
C08174=1050.994,437.837,366.981,175.870,43.062,158.607
C08175=1051.005,438.082,366.930,175.882,43.072,158.611
C08176=1051.016,438.327,366.879,175.896,43.083,158.615
C08177=1051.028,438.571,366.828,175.909,43.094,158.619
C08178=1051.039,438.815,366.778,175.922,43.105,158.623
C08179=1051.050,439.060,366.726,175.935,43.116,158.627
C08180=1051.061,439.305,366.675,175.947,43.127,158.631
C08181=1051.073,439.549,366.624,175.961,43.138,158.635
C08182=1051.084,439.793,366.573,175.974,43.149,158.639
C08183=1051.096,440.038,366.522,175.987,43.160,158.643
C08184=1051.106,440.282,366.471,176.001,43.171,158.647
C08185=1051.118,440.527,366.419,176.014,43.182,158.651
C08186=1051.130,440.771,366.368,176.027,43.193,158.656
C08187=1051.141,441.015,366.317,176.041,43.205,158.660
C08188=1051.153,441.260,366.265,176.054,43.216,158.664
C08189=1051.164,441.504,366.213,176.068,43.227,158.668
C08190=1051.176,441.749,366.162,176.081,43.239,158.673
C08191=1051.188,441.993,366.111,176.096,43.250,158.677
C08192=1051.199,442.237,366.058,176.109,43.261,158.681
C08193=1051.211,442.481,366.007,176.123,43.272,158.685
C08194=1051.223,442.726,365.955,176.136,43.284,158.690
C08195=1051.234,442.970,365.903,176.150,43.295,158.694
C08196=1051.246,443.215,365.851,176.165,43.307,158.699
C08197=1051.258,443.459,365.799,176.178,43.319,158.703
C08198=1051.269,443.703,365.748,176.192,43.330,158.707
C08199=1051.281,443.947,365.695,176.207,43.341,158.712
C08200=1051.294,444.191,365.643,176.220,43.353,158.716
C08201=1051.305,444.435,365.590,176.234,43.365,158.721
C08202=1051.317,444.679,365.538,176.249,43.377,158.725
C08203=1051.329,444.924,365.486,176.263,43.389,158.730
C08204=1051.341,445.168,365.434,176.278,43.400,158.734
C08205=1051.353,445.412,365.382,176.292,43.412,158.739
C08206=1051.365,445.655,365.328,176.307,43.424,158.743
C08207=1051.377,445.899,365.276,176.322,43.435,158.748
C08208=1051.389,446.143,365.224,176.336,43.448,158.752
C08209=1051.407,446.482,365.152,176.356,43.464,158.759
C08210=1051.426,446.822,365.081,176.377,43.480,158.765
C08211=1051.447,447.163,365.010,176.398,43.496,158.771
C08212=1051.470,447.504,364.940,176.419,43.511,158.777
C08213=1051.486,447.748,364.891,176.434,43.522,158.782
C08214=1051.503,447.992,364.843,176.449,43.533,158.786
C08215=1051.522,448.237,364.795,176.464,43.543,158.790
C08216=1051.541,448.482,364.748,176.480,43.554,158.795
C08217=1051.561,448.726,364.701,176.495,43.564,158.799
C08218=1051.581,448.971,364.655,176.510,43.574,158.803
C08219=1051.602,449.216,364.609,176.526,43.584,158.807
C08220=1051.624,449.461,364.564,176.542,43.594,158.811
C08221=1051.646,449.706,364.519,176.557,43.604,158.815
C08222=1051.669,449.952,364.475,176.574,43.613,158.819
C08223=1051.693,450.197,364.431,176.589,43.622,158.823
C08224=1051.718,450.442,364.388,176.605,43.632,158.827
C08225=1051.402,450.468,364.091,176.605,43.727,158.855
C08226=1051.378,450.222,364.134,176.588,43.717,158.851
C08227=1051.353,449.977,364.177,176.572,43.708,158.847
C08228=1051.329,449.732,364.221,176.557,43.699,158.843
C08229=1051.307,449.486,364.267,176.541,43.689,158.839
C08230=1051.285,449.241,364.312,176.525,43.679,158.834
C08231=1051.263,448.996,364.356,176.510,43.669,158.830
C08232=1051.243,448.751,364.403,176.494,43.659,158.826
C08233=1051.224,448.507,364.450,176.479,43.649,158.822
C08234=1051.205,448.262,364.497,176.463,43.639,158.818
C08235=1051.186,448.017,364.545,176.448,43.629,158.813
C08236=1051.168,447.773,364.594,176.432,43.618,158.809
C08237=1051.151,447.530,364.642,176.417,43.607,158.805
C08238=1051.131,447.206,364.708,176.397,43.593,158.799
C08239=1051.110,446.884,364.774,176.377,43.578,158.793
C08240=1051.091,446.562,364.842,176.358,43.563,158.787
C08241=1051.074,446.242,364.909,176.339,43.547,158.781
C08242=1051.061,445.998,364.961,176.324,43.536,158.776
C08243=1051.050,445.754,365.014,176.309,43.524,158.772
C08244=1051.037,445.511,365.067,176.295,43.512,158.767
C08245=1051.025,445.267,365.119,176.280,43.501,158.763
C08246=1051.013,445.023,365.171,176.266,43.489,158.758
C08247=1051.002,444.779,365.224,176.251,43.477,158.754
C08248=1050.989,444.535,365.276,176.237,43.465,158.749
C08249=1050.977,444.291,365.328,176.222,43.454,158.745
C08250=1050.965,444.046,365.381,176.208,43.442,158.740
C08251=1050.953,443.802,365.433,176.193,43.431,158.736
C08252=1050.941,443.558,365.485,176.180,43.419,158.731
C08253=1050.930,443.314,365.537,176.165,43.408,158.727
C08254=1050.918,443.069,365.589,176.151,43.396,158.723
C08255=1050.906,442.826,365.641,176.138,43.385,158.718
C08256=1050.895,442.581,365.693,176.124,43.373,158.714
C08257=1050.883,442.337,365.745,176.109,43.362,158.710
C08258=1050.871,442.093,365.796,176.096,43.351,158.705
C08259=1050.860,441.848,365.848,176.082,43.339,158.701
C08260=1050.848,441.604,365.899,176.069,43.328,158.697
C08261=1050.836,441.360,365.952,176.055,43.317,158.692
C08262=1050.825,441.116,366.003,176.042,43.306,158.688
C08263=1050.813,440.871,366.055,176.027,43.294,158.684
C08264=1050.801,440.626,366.106,176.014,43.284,158.680
C08265=1050.790,440.383,366.157,176.000,43.272,158.676
C08266=1050.779,440.138,366.208,175.987,43.262,158.672
C08267=1050.767,439.893,366.259,175.974,43.250,158.667
C08268=1050.756,439.649,366.311,175.960,43.239,158.663
C08269=1050.744,439.404,366.362,175.948,43.228,158.659
C08270=1050.733,439.160,366.413,175.935,43.218,158.655
C08271=1050.721,438.915,366.464,175.922,43.207,158.651
C08272=1050.710,438.672,366.515,175.908,43.196,158.647
C08273=1050.699,438.427,366.566,175.895,43.185,158.643
C08274=1050.688,438.182,366.617,175.882,43.174,158.639
C08275=1050.676,437.937,366.668,175.870,43.163,158.635
C08276=1050.665,437.693,366.718,175.857,43.153,158.631
C08277=1050.654,437.448,366.769,175.844,43.142,158.627
C08278=1050.643,437.204,366.820,175.831,43.132,158.623
C08279=1050.632,436.959,366.870,175.818,43.121,158.619
C08280=1050.621,436.715,366.921,175.805,43.110,158.615
C08281=1050.609,436.470,366.971,175.792,43.100,158.611
C08282=1050.598,436.225,367.022,175.781,43.089,158.607
C08283=1050.587,435.981,367.072,175.768,43.079,158.604
C08284=1050.576,435.735,367.122,175.756,43.068,158.600
C08285=1050.565,435.491,367.172,175.743,43.058,158.596
C08286=1050.553,435.247,367.222,175.731,43.047,158.592
C08287=1050.543,435.002,367.272,175.718,43.038,158.588
C08288=1050.532,434.757,367.322,175.706,43.027,158.585
C08289=1050.520,434.512,367.373,175.693,43.017,158.581
C08290=1050.509,434.267,367.422,175.682,43.006,158.577
C08291=1050.498,434.023,367.473,175.669,42.997,158.573
C08292=1050.487,433.778,367.522,175.657,42.986,158.569
C08293=1050.476,433.533,367.572,175.645,42.976,158.566
C08294=1050.457,433.122,367.656,175.624,42.959,158.560
C08295=1050.440,432.709,367.739,175.605,42.942,158.553
C08296=1050.422,432.297,367.822,175.585,42.925,158.547
C08297=1050.403,431.885,367.906,175.565,42.908,158.541
C08298=1050.393,431.641,367.955,175.554,42.898,158.538
C08299=1050.382,431.396,368.005,175.542,42.888,158.534
C08300=1050.372,431.151,368.054,175.531,42.879,158.531
C08301=1050.360,430.906,368.103,175.518,42.869,158.527
C08302=1050.351,430.661,368.152,175.507,42.859,158.523
C08303=1050.340,430.416,368.201,175.495,42.849,158.520
C08304=1050.329,430.171,368.251,175.484,42.839,158.516
C08305=1050.319,429.927,368.300,175.472,42.830,158.513
C08306=1050.308,429.681,368.348,175.461,42.820,158.509
C08307=1050.298,429.437,368.398,175.449,42.810,158.506
C08308=1050.288,429.191,368.447,175.438,42.801,158.502
C08309=1050.276,428.947,368.496,175.427,42.791,158.499
C08310=1050.266,428.702,368.544,175.415,42.781,158.496
C08311=1050.255,428.456,368.592,175.405,42.771,158.492
C08312=1050.245,428.212,368.642,175.394,42.762,158.489
C08313=1050.235,427.966,368.691,175.383,42.753,158.485
C08314=1050.224,427.722,368.738,175.371,42.743,158.482
C08315=1050.214,427.476,368.787,175.360,42.734,158.479
C08316=1050.204,427.231,368.835,175.349,42.725,158.475
C08317=1050.193,426.986,368.884,175.339,42.715,158.472
C08318=1050.183,426.741,368.932,175.328,42.706,158.469
C08319=1050.173,426.496,368.981,175.316,42.696,158.465
C08320=1050.162,426.251,369.029,175.305,42.687,158.462
C08321=1050.152,426.006,369.077,175.295,42.678,158.459
C08322=1050.142,425.761,369.125,175.284,42.668,158.456
C08323=1050.132,425.516,369.174,175.273,42.659,158.452
C08324=1050.121,425.271,369.222,175.263,42.650,158.449
C08325=1050.111,425.025,369.270,175.252,42.641,158.446
C08326=1050.101,424.780,369.318,175.241,42.632,158.443
C08327=1050.091,424.535,369.365,175.231,42.622,158.439
C08328=1050.079,424.290,369.413,175.220,42.614,158.436
C08329=1050.070,424.044,369.461,175.210,42.604,158.433
C08330=1050.060,423.824,369.505,175.201,42.597,158.430
C08331=1050.052,423.605,369.547,175.191,42.588,158.427
C08332=1050.042,423.384,369.589,175.182,42.581,158.425
C08333=1050.033,423.165,369.632,175.172,42.572,158.422
C08334=1050.024,422.944,369.676,175.163,42.565,158.419
C08335=1050.015,422.724,369.718,175.154,42.556,158.416
C08336=1050.006,422.504,369.760,175.145,42.548,158.413
C08337=1049.997,422.284,369.803,175.135,42.540,158.411
C08338=1049.987,422.039,369.851,175.125,42.532,158.408
C08339=1049.977,421.793,369.898,175.115,42.523,158.405
C08340=1049.967,421.548,369.946,175.105,42.514,158.402
C08341=1049.957,421.303,369.993,175.095,42.505,158.399
C08342=1049.946,421.058,370.040,175.084,42.496,158.395
C08343=1049.937,420.812,370.088,175.074,42.488,158.392
C08344=1049.928,420.567,370.134,175.065,42.479,158.390
C08345=1049.918,420.321,370.181,175.054,42.470,158.386
C08346=1049.907,420.076,370.228,175.044,42.462,158.383
C08347=1049.898,419.831,370.276,175.035,42.453,158.381
C08348=1049.888,419.585,370.323,175.025,42.444,158.377
C08349=1049.878,419.340,370.370,175.014,42.436,158.375
C08350=1049.870,419.120,370.412,175.006,42.428,158.372
C08351=1049.861,418.901,370.454,174.997,42.421,158.369
C08352=1049.852,418.681,370.495,174.989,42.413,158.367
C08353=1049.843,418.462,370.538,174.979,42.405,158.364
C08354=1049.834,418.242,370.580,174.971,42.398,158.362
C08355=1049.825,418.022,370.621,174.962,42.391,158.359
C08356=1049.816,417.803,370.663,174.954,42.383,158.356
C08357=1049.808,417.583,370.705,174.945,42.375,158.354
C08358=1049.798,417.338,370.751,174.935,42.367,158.351
C08359=1049.789,417.092,370.798,174.926,42.359,158.348
C08360=1049.779,416.847,370.844,174.916,42.351,158.345
C08361=1049.768,416.602,370.890,174.907,42.342,158.342
C08362=1049.758,416.356,370.937,174.897,42.334,158.340
C08363=1049.749,416.111,370.983,174.888,42.325,158.337
C08364=1049.739,415.865,371.029,174.878,42.318,158.334
C08365=1049.730,415.619,371.076,174.869,42.309,158.331
C08366=1049.720,415.374,371.122,174.860,42.301,158.329
C08367=1049.711,415.128,371.168,174.850,42.293,158.326
C08368=1049.702,414.883,371.214,174.841,42.285,158.323
C08369=1049.692,414.637,371.260,174.832,42.277,158.320
C08370=1049.683,414.391,371.306,174.823,42.268,158.317
C08371=1049.673,414.145,371.353,174.814,42.260,158.315
C08372=1049.664,413.900,371.399,174.805,42.253,158.312
C08373=1049.655,413.654,371.444,174.795,42.245,158.309
C08374=1049.645,413.410,371.490,174.786,42.236,158.307
C08375=1049.635,413.164,371.536,174.777,42.228,158.304
C08376=1049.626,412.918,371.582,174.768,42.220,158.301
C08377=1049.616,412.673,371.628,174.759,42.213,158.299
C08378=1049.607,412.426,371.674,174.750,42.205,158.296
C08379=1049.597,412.181,371.719,174.741,42.197,158.293
C08380=1049.588,411.935,371.765,174.731,42.189,158.291
C08381=1049.578,411.690,371.809,174.723,42.181,158.288
C08382=1049.569,411.443,371.855,174.714,42.174,158.285
C08383=1049.559,411.198,371.901,174.705,42.166,158.283
C08384=1049.550,410.953,371.946,174.696,42.158,158.280
C08385=1049.541,410.707,371.992,174.688,42.150,158.278
C08386=1049.531,410.461,372.036,174.679,42.143,158.275
C08387=1049.522,410.215,372.082,174.670,42.135,158.273
C08388=1049.512,409.970,372.127,174.661,42.127,158.270
C08389=1049.503,409.724,372.172,174.652,42.120,158.267
C08390=1049.494,409.478,372.218,174.643,42.112,158.265
C08391=1049.484,409.232,372.263,174.635,42.105,158.262
C08392=1049.475,408.986,372.308,174.626,42.097,158.260
C08393=1049.465,408.741,372.353,174.618,42.089,158.257
C08394=1049.457,408.496,372.398,174.609,42.082,158.255
C08395=1049.447,408.250,372.443,174.601,42.074,158.252
C08396=1049.438,408.004,372.488,174.592,42.067,158.250
C08397=1049.429,407.758,372.532,174.584,42.059,158.247
C08398=1049.420,407.512,372.578,174.575,42.052,158.245
C08399=1049.411,407.266,372.623,174.567,42.044,158.242
C08400=1049.401,407.020,372.667,174.558,42.037,158.240
C08401=1049.392,406.775,372.713,174.550,42.030,158.238
C08402=1049.383,406.530,372.757,174.541,42.022,158.235
C08403=1049.375,406.283,372.802,174.533,42.014,158.233
C08404=1049.365,406.038,372.847,174.524,42.008,158.230
C08405=1049.356,405.791,372.891,174.516,42.000,158.228
C08406=1049.347,405.547,372.936,174.509,41.993,158.226
C08407=1049.338,405.300,372.981,174.500,41.985,158.223
C08408=1049.329,405.054,373.025,174.492,41.978,158.221
C08409=1049.321,404.809,373.070,174.483,41.971,158.218
C08410=1049.306,404.427,373.139,174.471,41.960,158.215
C08411=1049.292,404.044,373.208,174.458,41.949,158.211
C08412=1049.279,403.662,373.276,174.446,41.938,158.207
C08413=1049.264,403.280,373.345,174.433,41.927,158.204
C08414=1049.255,403.034,373.389,174.425,41.919,158.201
C08415=1049.246,402.788,373.433,174.417,41.912,158.199
C08416=1049.238,402.543,373.477,174.408,41.905,158.197
C08417=1049.229,402.296,373.522,174.401,41.898,158.194
C08418=1049.220,402.051,373.565,174.393,41.891,158.192
C08419=1049.210,401.805,373.609,174.385,41.884,158.190
C08420=1049.202,401.559,373.654,174.377,41.877,158.188
C08421=1049.193,401.312,373.697,174.369,41.870,158.185
C08422=1049.184,401.067,373.741,174.361,41.864,158.183
C08423=1049.175,400.821,373.785,174.353,41.856,158.181
C08424=1049.166,400.575,373.829,174.346,41.849,158.179
C08425=1049.158,400.329,373.872,174.338,41.843,158.176
C08426=1049.148,400.083,373.916,174.329,41.836,158.174
C08427=1049.140,399.837,373.959,174.322,41.829,158.172
C08428=1049.130,399.591,374.003,174.314,41.822,158.170
C08429=1049.122,399.345,374.046,174.306,41.815,158.168
C08430=1049.114,399.099,374.090,174.299,41.808,158.165
C08431=1049.105,398.853,374.133,174.291,41.802,158.163
C08432=1049.096,398.607,374.177,174.284,41.795,158.161
C08433=1049.087,398.361,374.221,174.276,41.789,158.159
C08434=1049.079,398.115,374.264,174.267,41.782,158.157
C08435=1049.070,397.869,374.307,174.260,41.775,158.154
C08436=1049.061,397.623,374.351,174.252,41.768,158.152
C08437=1049.052,397.377,374.394,174.245,41.762,158.150
C08438=1049.044,397.131,374.437,174.237,41.755,158.148
C08439=1049.035,396.885,374.480,174.230,41.749,158.146
C08440=1049.027,396.639,374.523,174.222,41.742,158.144
C08441=1049.018,396.393,374.567,174.215,41.735,158.142
C08442=1049.010,396.147,374.610,174.207,41.729,158.140
C08443=1049.001,395.900,374.653,174.200,41.722,158.138
C08444=1048.991,395.654,374.695,174.192,41.716,158.135
C08445=1048.983,395.408,374.738,174.185,41.709,158.133
C08446=1048.974,395.162,374.781,174.177,41.702,158.131
C08447=1048.966,394.916,374.824,174.170,41.696,158.129
C08448=1048.957,394.670,374.867,174.163,41.690,158.127
C08449=1048.949,394.424,374.911,174.155,41.683,158.125
C08450=1048.940,394.178,374.953,174.149,41.677,158.123
C08451=1048.931,393.932,374.996,174.141,41.670,158.121
C08452=1048.923,393.686,375.038,174.134,41.664,158.119
C08453=1048.914,393.440,375.081,174.127,41.658,158.117
C08454=1048.906,393.194,375.124,174.119,41.651,158.115
C08455=1048.897,392.948,375.167,174.112,41.645,158.113
C08456=1048.889,392.702,375.209,174.105,41.639,158.111
C08457=1048.881,392.456,375.252,174.097,41.632,158.109
C08458=1048.872,392.210,375.295,174.091,41.626,158.107
C08459=1048.863,391.963,375.336,174.084,41.620,158.105
C08460=1048.855,391.717,375.380,174.076,41.613,158.103
C08461=1048.846,391.471,375.422,174.069,41.607,158.101
C08462=1048.837,391.224,375.464,174.062,41.601,158.099
C08463=1048.830,390.979,375.506,174.054,41.595,158.097
C08464=1048.821,390.732,375.549,174.048,41.589,158.095
C08465=1048.812,390.487,375.591,174.041,41.583,158.093
C08466=1048.800,390.123,375.653,174.030,41.573,158.090
C08467=1048.788,389.759,375.716,174.020,41.564,158.087
C08468=1048.775,389.396,375.778,174.010,41.555,158.084
C08469=1048.763,389.033,375.840,173.999,41.546,158.082
C08470=1048.754,388.787,375.882,173.992,41.540,158.080
C08471=1048.746,388.540,375.924,173.985,41.534,158.078
C08472=1048.737,388.294,375.966,173.979,41.528,158.076
C08473=1048.729,388.048,376.007,173.972,41.522,158.074
C08474=1048.721,387.801,376.049,173.964,41.516,158.072
C08475=1048.712,387.555,376.091,173.958,41.510,158.070
C08476=1048.704,387.309,376.132,173.951,41.504,158.068
C08477=1048.695,387.063,376.175,173.944,41.499,158.067
C08478=1048.687,386.816,376.216,173.938,41.492,158.065
C08479=1048.679,386.570,376.258,173.931,41.487,158.063
C08480=1048.670,386.323,376.299,173.923,41.481,158.061
C08481=1048.662,386.078,376.341,173.917,41.475,158.059
C08482=1048.654,385.830,376.382,173.910,41.469,158.057
C08483=1048.646,385.585,376.424,173.903,41.463,158.055
C08484=1048.637,385.338,376.465,173.897,41.458,158.054
C08485=1048.629,385.092,376.507,173.890,41.451,158.052
C08486=1048.620,384.845,376.548,173.884,41.446,158.050
C08487=1048.612,384.600,376.590,173.877,41.440,158.048
C08488=1048.604,384.352,376.631,173.869,41.434,158.046
C08489=1048.596,384.107,376.673,173.863,41.428,158.044
C08490=1048.587,383.860,376.714,173.856,41.423,158.043
C08491=1048.580,383.614,376.756,173.850,41.417,158.041
C08492=1048.572,383.367,376.796,173.843,41.411,158.039
C08493=1048.563,383.121,376.838,173.837,41.406,158.037
C08494=1048.555,382.875,376.879,173.830,41.400,158.036
C08495=1048.547,382.628,376.921,173.824,41.394,158.034
C08496=1048.538,382.382,376.961,173.817,41.388,158.032
C08497=1048.531,382.135,377.003,173.811,41.382,158.030
C08498=1048.522,381.889,377.044,173.804,41.377,158.028
C08499=1048.514,381.643,377.085,173.798,41.371,158.027
C08500=1048.506,381.396,377.126,173.791,41.366,158.025
C08501=1048.499,381.150,377.167,173.785,41.360,158.023
C08502=1048.490,380.903,377.208,173.778,41.355,158.022
C08503=1048.482,380.657,377.249,173.772,41.349,158.020
C08504=1048.475,380.411,377.290,173.766,41.343,158.018
C08505=1048.467,380.164,377.331,173.759,41.338,158.016
C08506=1048.459,379.918,377.372,173.753,41.332,158.015
C08507=1048.450,379.671,377.413,173.746,41.327,158.013
C08508=1048.443,379.424,377.454,173.740,41.321,158.011
C08509=1048.434,379.178,377.494,173.734,41.316,158.010
C08510=1048.426,378.932,377.535,173.727,41.310,158.008
C08511=1048.417,378.685,377.576,173.721,41.305,158.006
C08512=1048.410,378.438,377.616,173.714,41.299,158.004
C08513=1048.402,378.192,377.656,173.709,41.294,158.003
C08514=1048.394,377.946,377.697,173.703,41.289,158.001
C08515=1048.386,377.699,377.737,173.696,41.283,158.000
C08516=1048.377,377.453,377.778,173.690,41.278,157.998
C08517=1048.370,377.206,377.818,173.684,41.272,157.996
C08518=1048.361,376.959,377.859,173.677,41.267,157.995
C08519=1048.353,376.713,377.900,173.671,41.262,157.993
C08520=1048.345,376.466,377.940,173.665,41.256,157.991
C08521=1048.337,376.220,377.980,173.659,41.251,157.990
C08522=1048.327,375.889,378.034,173.651,41.244,157.987
C08523=1048.316,375.559,378.088,173.643,41.237,157.985
C08524=1048.306,375.228,378.142,173.634,41.230,157.983
C08525=1048.295,374.898,378.196,173.626,41.223,157.981
C08526=1048.287,374.651,378.236,173.620,41.218,157.979
C08527=1048.279,374.405,378.276,173.614,41.212,157.978
C08528=1048.271,374.158,378.316,173.608,41.207,157.976
C08529=1048.264,373.911,378.356,173.601,41.202,157.975
C08530=1048.256,373.665,378.397,173.596,41.197,157.973
C08531=1048.248,373.418,378.437,173.590,41.192,157.971
C08532=1048.240,373.171,378.477,173.584,41.186,157.970
C08533=1048.232,372.925,378.517,173.577,41.181,157.968
C08534=1048.225,372.679,378.557,173.571,41.176,157.967
C08535=1048.217,372.432,378.596,173.566,41.171,157.965
C08536=1048.209,372.185,378.636,173.560,41.166,157.964
C08537=1048.201,371.938,378.676,173.554,41.161,157.962
C08538=1048.193,371.692,378.716,173.549,41.156,157.961
C08539=1048.185,371.445,378.756,173.542,41.151,157.959
C08540=1048.178,371.199,378.796,173.536,41.146,157.957
C08541=1048.170,370.952,378.835,173.530,41.140,157.956
C08542=1048.162,370.705,378.875,173.525,41.136,157.954
C08543=1048.154,370.458,378.915,173.519,41.130,157.953
C08544=1048.146,370.212,378.954,173.513,41.126,157.951
C08545=1048.139,369.965,378.993,173.507,41.120,157.950
C08546=1048.131,369.718,379.033,173.501,41.116,157.948
C08547=1048.123,369.472,379.073,173.495,41.111,157.947
C08548=1048.115,369.225,379.112,173.489,41.106,157.945
C08549=1048.107,368.978,379.152,173.484,41.101,157.944
C08550=1048.100,368.731,379.191,173.478,41.096,157.942
C08551=1048.092,368.485,379.230,173.472,41.091,157.941
C08552=1048.084,368.238,379.270,173.467,41.086,157.939
C08553=1048.076,367.992,379.309,173.461,41.081,157.938
C08554=1048.069,367.744,379.348,173.455,41.076,157.936
C08555=1048.061,367.497,379.388,173.450,41.072,157.935
C08556=1048.053,367.252,379.427,173.443,41.066,157.933
C08557=1048.046,367.004,379.466,173.437,41.062,157.932
C08558=1048.037,366.757,379.505,173.432,41.057,157.931
C08559=1048.030,366.511,379.544,173.426,41.052,157.929
C08560=1048.022,366.264,379.584,173.420,41.047,157.928
C08561=1048.015,366.017,379.622,173.415,41.042,157.926
C08562=1048.007,365.771,379.662,173.409,41.038,157.925
C08563=1047.999,365.523,379.701,173.404,41.033,157.923
C08564=1047.992,365.277,379.741,173.398,41.028,157.922
C08565=1047.984,365.030,379.779,173.392,41.023,157.920
C08566=1047.977,364.783,379.818,173.387,41.018,157.919
C08567=1047.969,364.536,379.857,173.381,41.014,157.917
C08568=1047.962,364.289,379.896,173.376,41.009,157.916
C08569=1047.954,364.042,379.935,173.370,41.004,157.915
C08570=1047.947,363.796,379.974,173.364,41.000,157.913
C08571=1047.938,363.549,380.013,173.360,40.995,157.912
C08572=1047.932,363.302,380.052,173.354,40.990,157.910
C08573=1047.924,363.055,380.090,173.349,40.985,157.909
C08574=1047.916,362.808,380.130,173.343,40.981,157.908
C08575=1047.909,362.562,380.168,173.338,40.976,157.906
C08576=1047.901,362.315,380.207,173.332,40.971,157.905
C08577=1047.894,362.068,380.246,173.326,40.967,157.903
C08578=1047.884,361.756,380.294,173.319,40.961,157.902
C08579=1047.874,361.445,380.343,173.313,40.955,157.900
C08580=1047.864,361.134,380.391,173.306,40.949,157.898
C08581=1047.855,360.822,380.439,173.299,40.944,157.896
C08582=1047.847,360.576,380.478,173.293,40.939,157.895
C08583=1047.839,360.328,380.516,173.288,40.935,157.894
C08584=1047.832,360.082,380.555,173.283,40.930,157.892
C08585=1047.825,359.835,380.593,173.278,40.925,157.891
C08586=1047.817,359.588,380.632,173.272,40.921,157.890
C08587=1047.809,359.341,380.670,173.267,40.916,157.888
C08588=1047.802,359.094,380.708,173.261,40.912,157.887
C08589=1047.795,358.847,380.747,173.256,40.907,157.886
C08590=1047.787,358.600,380.785,173.250,40.903,157.884
C08591=1047.779,358.354,380.823,173.246,40.898,157.883
C08592=1047.772,358.107,380.861,173.240,40.894,157.882
C08593=1047.764,357.859,380.900,173.235,40.889,157.880
C08594=1047.757,357.613,380.938,173.230,40.885,157.879
C08595=1047.750,357.365,380.976,173.224,40.881,157.878
C08596=1047.742,357.119,381.014,173.220,40.876,157.876
C08597=1047.735,356.871,381.052,173.214,40.872,157.875
C08598=1047.727,356.625,381.090,173.209,40.867,157.874
C08599=1047.720,356.377,381.128,173.203,40.863,157.873
C08600=1047.712,356.131,381.166,173.198,40.859,157.871
C08601=1047.705,355.884,381.204,173.193,40.854,157.870
C08602=1047.697,355.637,381.242,173.188,40.850,157.869
C08603=1047.690,355.389,381.280,173.183,40.846,157.867
C08604=1047.682,355.142,381.317,173.177,40.841,157.866
C08605=1047.675,354.896,381.356,173.172,40.837,157.865
C08606=1047.668,354.649,381.393,173.167,40.833,157.864
C08607=1047.660,354.402,381.431,173.162,40.829,157.862
C08608=1047.652,354.154,381.469,173.157,40.824,157.861
C08609=1047.645,353.907,381.507,173.152,40.819,157.860
C08610=1047.638,353.660,381.544,173.147,40.815,157.858
C08611=1047.630,353.413,381.583,173.141,40.811,157.857
C08612=1047.623,353.166,381.620,173.136,40.807,157.856
C08613=1047.616,352.919,381.658,173.132,40.803,157.855
C08614=1047.608,352.672,381.695,173.126,40.798,157.853
C08615=1047.601,352.425,381.733,173.121,40.794,157.852
C08616=1047.594,352.178,381.770,173.117,40.790,157.851
C08617=1047.586,351.932,381.808,173.111,40.786,157.850
C08618=1047.578,351.684,381.845,173.106,40.782,157.848
C08619=1047.571,351.437,381.883,173.101,40.777,157.847
C08620=1047.564,351.190,381.920,173.096,40.773,157.846
C08621=1047.557,350.943,381.958,173.091,40.769,157.845
C08622=1047.549,350.696,381.995,173.086,40.765,157.843
C08623=1047.542,350.449,382.033,173.081,40.760,157.842
C08624=1047.535,350.202,382.071,173.076,40.756,157.841
C08625=1047.527,349.954,382.107,173.071,40.752,157.840
C08626=1047.520,349.707,382.144,173.066,40.748,157.839
C08627=1047.513,349.460,382.182,173.061,40.744,157.837
C08628=1047.506,349.213,382.219,173.056,40.740,157.836
C08629=1047.498,348.966,382.256,173.051,40.736,157.835
C08630=1047.490,348.719,382.294,173.047,40.731,157.834
C08631=1047.483,348.471,382.331,173.042,40.728,157.833
C08632=1047.476,348.225,382.367,173.036,40.724,157.831
C08633=1047.469,347.978,382.405,173.032,40.719,157.830
C08634=1047.460,347.672,382.450,173.025,40.715,157.829
C08635=1047.450,347.366,382.496,173.020,40.709,157.827
C08636=1047.442,347.060,382.543,173.013,40.705,157.826
C08637=1047.433,346.754,382.588,173.007,40.699,157.824
C08638=1047.425,346.507,382.625,173.002,40.696,157.823
C08639=1047.418,346.260,382.662,172.998,40.691,157.822
C08640=1047.411,346.013,382.699,172.993,40.688,157.821
C08641=1047.403,345.766,382.736,172.988,40.683,157.820
C08642=1047.396,345.518,382.773,172.983,40.679,157.818
C08643=1047.389,345.271,382.810,172.979,40.675,157.817
C08644=1047.382,345.024,382.846,172.974,40.671,157.816
C08645=1047.375,344.777,382.883,172.969,40.667,157.815
C08646=1047.367,344.530,382.920,172.964,40.663,157.814
C08647=1047.360,344.282,382.957,172.960,40.659,157.813
C08648=1047.354,344.035,382.994,172.955,40.656,157.812
C08649=1047.346,343.788,383.030,172.950,40.651,157.810
C08650=1047.339,343.540,383.067,172.945,40.648,157.809
C08651=1047.332,343.294,383.103,172.941,40.643,157.808
C08652=1047.325,343.046,383.140,172.936,40.640,157.807
C08653=1047.317,342.799,383.176,172.932,40.636,157.806
C08654=1047.310,342.552,383.214,172.926,40.632,157.805
C08655=1047.303,342.305,383.250,172.922,40.628,157.804
C08656=1047.296,342.057,383.286,172.917,40.625,157.803
C08657=1047.288,341.810,383.323,172.913,40.620,157.801
C08658=1047.282,341.563,383.359,172.907,40.617,157.800
C08659=1047.274,341.315,383.395,172.903,40.613,157.799
C08660=1047.266,341.068,383.432,172.898,40.609,157.798
C08661=1047.260,340.821,383.468,172.894,40.605,157.797
C08662=1047.252,340.574,383.505,172.889,40.601,157.796
C08663=1047.245,340.327,383.541,172.884,40.597,157.795
C08664=1047.238,340.080,383.578,172.880,40.594,157.794
C08665=1047.230,339.832,383.614,172.875,40.590,157.793
C08666=1047.223,339.585,383.650,172.871,40.586,157.792
C08667=1047.216,339.338,383.686,172.866,40.583,157.790
C08668=1047.210,339.090,383.722,172.861,40.578,157.789
C08669=1047.202,338.843,383.758,172.856,40.575,157.788
C08670=1047.196,338.596,383.794,172.852,40.571,157.787
C08671=1047.188,338.348,383.831,172.848,40.567,157.786
C08672=1047.180,338.101,383.867,172.843,40.563,157.785
C08673=1047.174,337.854,383.903,172.839,40.560,157.784
C08674=1047.166,337.606,383.939,172.834,40.556,157.783
C08675=1047.159,337.359,383.975,172.829,40.552,157.782
C08676=1047.152,337.111,384.011,172.825,40.548,157.781
C08677=1047.145,336.864,384.047,172.820,40.545,157.780
C08678=1047.138,336.618,384.083,172.816,40.541,157.778
C08679=1047.131,336.370,384.119,172.812,40.537,157.777
C08680=1047.125,336.123,384.155,172.807,40.534,157.776
C08681=1047.117,335.875,384.191,172.802,40.530,157.775
C08682=1047.110,335.628,384.226,172.798,40.526,157.774
C08683=1047.102,335.380,384.263,172.793,40.522,157.773
C08684=1047.095,335.134,384.298,172.789,40.519,157.772
C08685=1047.088,334.886,384.334,172.785,40.515,157.771
C08686=1047.081,334.639,384.370,172.780,40.512,157.770
C08687=1047.074,334.391,384.405,172.776,40.508,157.769
C08688=1047.067,334.144,384.441,172.772,40.504,157.768
C08689=1047.060,333.897,384.476,172.767,40.501,157.767
C08690=1047.051,333.587,384.521,172.761,40.496,157.766
C08691=1047.042,333.277,384.566,172.756,40.492,157.764
C08692=1047.034,332.968,384.610,172.750,40.487,157.763
C08693=1047.024,332.659,384.655,172.745,40.483,157.762
C08694=1047.017,332.411,384.691,172.740,40.479,157.761
C08695=1047.010,332.163,384.726,172.736,40.476,157.760
C08696=1047.003,331.916,384.762,172.732,40.472,157.759
C08697=1046.996,331.668,384.798,172.728,40.468,157.758
C08698=1046.990,331.421,384.833,172.723,40.465,157.757
C08699=1046.983,331.174,384.869,172.719,40.462,157.756
C08700=1046.976,330.927,384.904,172.714,40.458,157.755
C08701=1046.968,330.678,384.939,172.710,40.455,157.754
C08702=1046.962,330.431,384.974,172.705,40.451,157.753
C08703=1046.955,330.184,385.010,172.701,40.447,157.752
C08704=1046.948,329.937,385.045,172.697,40.444,157.751
C08705=1046.940,329.689,385.081,172.693,40.440,157.750
C08706=1046.934,329.442,385.116,172.688,40.437,157.749
C08707=1046.926,329.195,385.151,172.684,40.433,157.748
C08708=1046.919,328.946,385.186,172.680,40.430,157.747
C08709=1046.912,328.699,385.221,172.676,40.426,157.746
C08710=1046.905,328.452,385.256,172.671,40.423,157.745
C08711=1046.898,328.205,385.291,172.667,40.420,157.744
C08712=1046.890,327.957,385.326,172.663,40.416,157.743
C08713=1046.883,327.710,385.361,172.659,40.413,157.742
C08714=1046.876,327.462,385.396,172.655,40.410,157.741
C08715=1046.869,327.215,385.431,172.650,40.406,157.740
C08716=1046.861,326.967,385.466,172.646,40.403,157.739
C08717=1046.854,326.720,385.501,172.642,40.399,157.738
C08718=1046.847,326.472,385.535,172.638,40.396,157.737
C08719=1046.840,326.225,385.570,172.633,40.393,157.736
C08720=1046.833,325.978,385.605,172.629,40.389,157.735
C08721=1046.826,325.730,385.640,172.625,40.386,157.734
C08722=1046.819,325.482,385.675,172.621,40.382,157.733
C08723=1046.812,325.235,385.709,172.617,40.379,157.732
C08724=1046.805,324.987,385.744,172.613,40.376,157.731
C08725=1046.797,324.740,385.779,172.608,40.372,157.730
C08726=1046.791,324.493,385.814,172.604,40.369,157.729
C08727=1046.784,324.245,385.848,172.600,40.366,157.728
C08728=1046.777,323.998,385.883,172.596,40.363,157.728
C08729=1046.770,323.750,385.918,172.592,40.359,157.726
C08730=1046.763,323.503,385.952,172.588,40.355,157.726
C08731=1046.756,323.255,385.987,172.584,40.352,157.725
C08732=1046.749,323.008,386.022,172.579,40.349,157.724
C08733=1046.742,322.760,386.056,172.575,40.346,157.723
C08734=1046.735,322.513,386.091,172.571,40.343,157.722
C08735=1046.728,322.265,386.125,172.567,40.339,157.721
C08736=1046.721,322.018,386.160,172.563,40.336,157.720
C08737=1046.714,321.771,386.195,172.559,40.332,157.719
C08738=1046.707,321.523,386.229,172.555,40.329,157.718
C08739=1046.700,321.275,386.264,172.551,40.326,157.717
C08740=1046.693,321.028,386.298,172.547,40.323,157.716
C08741=1046.686,320.780,386.333,172.543,40.320,157.715
C08742=1046.679,320.533,386.367,172.538,40.316,157.715
C08743=1046.673,320.285,386.401,172.534,40.313,157.713
C08744=1046.665,320.038,386.436,172.530,40.309,157.713
C08745=1046.659,319.790,386.470,172.526,40.306,157.712
C08746=1046.650,319.475,386.514,172.521,40.302,157.711
C08747=1046.642,319.161,386.558,172.517,40.298,157.709
C08748=1046.632,318.847,386.601,172.511,40.294,157.708
C08749=1046.623,318.531,386.645,172.506,40.290,157.707
C08750=1046.617,318.284,386.680,172.502,40.287,157.706
C08751=1046.610,318.037,386.713,172.498,40.283,157.705
C08752=1046.604,317.789,386.748,172.494,40.280,157.704
C08753=1046.596,317.541,386.782,172.490,40.276,157.703
C08754=1046.590,317.294,386.817,172.486,40.273,157.702
C08755=1046.583,317.047,386.850,172.482,40.270,157.702
C08756=1046.577,316.799,386.885,172.479,40.267,157.701
C08757=1046.569,316.551,386.919,172.475,40.264,157.700
C08758=1046.563,316.303,386.953,172.471,40.261,157.699
C08759=1046.555,316.056,386.987,172.467,40.258,157.698
C08760=1046.550,315.809,387.022,172.463,40.254,157.697
C08761=1046.542,315.561,387.055,172.459,40.251,157.696
C08762=1046.536,315.313,387.090,172.455,40.248,157.695
C08763=1046.529,315.066,387.123,172.451,40.245,157.694
C08764=1046.523,314.818,387.158,172.447,40.241,157.694
C08765=1046.516,314.571,387.191,172.443,40.238,157.693
C08766=1046.509,314.323,387.226,172.439,40.235,157.692
C08767=1046.503,314.076,387.259,172.435,40.232,157.691
C08768=1046.496,313.828,387.294,172.431,40.228,157.690
C08769=1046.489,313.581,387.328,172.427,40.225,157.689
C08770=1046.483,313.333,387.362,172.423,40.222,157.688
C08771=1046.476,313.085,387.395,172.420,40.219,157.687
C08772=1046.470,312.838,387.430,172.416,40.216,157.686
C08773=1046.463,312.590,387.463,172.412,40.213,157.686
C08774=1046.456,312.342,387.497,172.409,40.209,157.685
C08775=1046.448,312.095,387.531,172.405,40.207,157.684
C08776=1046.442,311.848,387.564,172.401,40.203,157.683
C08777=1046.435,311.599,387.598,172.397,40.200,157.682
C08778=1046.428,311.352,387.631,172.393,40.197,157.681
C08779=1046.420,311.105,387.664,172.389,40.194,157.680
C08780=1046.413,310.857,387.698,172.386,40.192,157.680
C08781=1046.406,310.609,387.731,172.382,40.188,157.679
C08782=1046.399,310.361,387.765,172.378,40.186,157.678
C08783=1046.392,310.114,387.798,172.374,40.182,157.677
C08784=1046.386,309.866,387.832,172.370,40.179,157.676
C08785=1046.379,309.619,387.865,172.366,40.176,157.676
C08786=1046.372,309.371,387.898,172.362,40.173,157.675
C08787=1046.365,309.123,387.932,172.359,40.170,157.674
C08788=1046.358,308.876,387.965,172.355,40.167,157.673
C08789=1046.351,308.628,387.998,172.351,40.165,157.672
C08790=1046.343,308.381,388.032,172.347,40.161,157.671
C08791=1046.337,308.133,388.065,172.344,40.159,157.671
C08792=1046.330,307.885,388.098,172.340,40.155,157.670
C08793=1046.324,307.638,388.131,172.336,40.153,157.669
C08794=1046.316,307.390,388.165,172.332,40.149,157.668
C08795=1046.310,307.142,388.198,172.329,40.147,157.667
C08796=1046.303,306.895,388.231,172.325,40.143,157.666
C08797=1046.297,306.647,388.264,172.321,40.141,157.666
C08798=1046.289,306.400,388.297,172.317,40.137,157.665
C08799=1046.282,306.152,388.330,172.314,40.135,157.664
C08800=1046.276,305.904,388.363,172.310,40.131,157.663
C08801=1046.269,305.657,388.397,172.307,40.129,157.662
C08802=1046.260,305.347,388.438,172.302,40.125,157.661
C08803=1046.252,305.036,388.480,172.297,40.121,157.660
C08804=1046.244,304.727,388.521,172.292,40.117,157.659
C08805=1046.235,304.416,388.562,172.288,40.114,157.658
C08806=1046.228,304.168,388.596,172.285,40.111,157.657
C08807=1046.222,303.921,388.628,172.281,40.108,157.657
C08808=1046.215,303.673,388.662,172.277,40.105,157.656
C08809=1046.207,303.426,388.694,172.273,40.102,157.655
C08810=1046.201,303.178,388.727,172.270,40.099,157.654
C08811=1046.194,302.930,388.760,172.266,40.096,157.653
C08812=1046.188,302.682,388.793,172.263,40.093,157.653
C08813=1046.181,302.434,388.826,172.259,40.090,157.652
C08814=1046.175,302.187,388.859,172.255,40.087,157.651
C08815=1046.167,301.940,388.892,172.252,40.085,157.650
C08816=1046.160,301.692,388.925,172.248,40.081,157.649
C08817=1046.154,301.444,388.958,172.244,40.079,157.649
C08818=1046.148,301.196,388.990,172.241,40.076,157.648
C08819=1046.141,300.948,389.023,172.238,40.073,157.647
C08820=1046.134,300.701,389.056,172.234,40.070,157.646
C08821=1046.128,300.453,389.088,172.230,40.067,157.645
C08822=1046.121,300.205,389.121,172.226,40.064,157.645
C08823=1046.114,299.957,389.154,172.224,40.061,157.644
C08824=1046.108,299.710,389.187,172.220,40.058,157.643
C08825=1046.102,299.462,389.220,172.216,40.055,157.642
C08826=1046.094,299.214,389.252,172.213,40.052,157.641
C08827=1046.088,298.967,389.285,172.209,40.049,157.641
C08828=1046.082,298.719,389.318,172.205,40.046,157.640
C08829=1046.075,298.471,389.350,172.202,40.044,157.639
C08830=1046.068,298.223,389.384,172.199,40.040,157.638
C08831=1046.061,297.976,389.416,172.195,40.038,157.637
C08832=1046.055,297.728,389.448,172.191,40.035,157.637
C08833=1046.049,297.481,389.481,172.188,40.032,157.636
C08834=1046.042,297.232,389.514,172.185,40.029,157.635
C08835=1046.035,296.985,389.546,172.181,40.026,157.634
C08836=1046.029,296.738,389.579,172.178,40.023,157.634
C08837=1046.023,296.489,389.611,172.174,40.020,157.633
C08838=1046.016,296.242,389.644,172.170,40.017,157.632
C08839=1046.010,295.994,389.677,172.168,40.015,157.631
C08840=1046.002,295.746,389.709,172.164,40.012,157.631
C08841=1045.996,295.498,389.741,172.160,40.009,157.630
C08842=1045.989,295.251,389.773,172.156,40.006,157.629
C08843=1045.983,295.003,389.806,172.153,40.003,157.628
C08844=1045.976,294.754,389.838,172.150,40.000,157.627
C08845=1045.969,294.507,389.871,172.146,39.998,157.627
C08846=1045.962,294.260,389.903,172.143,39.995,157.626
C08847=1045.956,294.012,389.934,172.139,39.992,157.625
C08848=1045.949,293.764,389.967,172.136,39.990,157.624
C08849=1045.943,293.516,389.998,172.133,39.987,157.624
C08850=1045.936,293.268,390.032,172.129,39.984,157.623
C08851=1045.929,293.021,390.064,172.125,39.981,157.622
C08852=1045.922,292.773,390.095,172.122,39.978,157.621
C08853=1045.916,292.525,390.128,172.119,39.975,157.621
C08854=1045.909,292.277,390.159,172.116,39.972,157.620
C08855=1045.902,292.029,390.191,172.112,39.970,157.619
C08856=1045.895,291.781,390.224,172.108,39.967,157.618
C08857=1045.889,291.533,390.255,172.106,39.964,157.618
C08858=1045.881,291.240,390.294,172.102,39.961,157.617
C08859=1045.873,290.946,390.331,172.097,39.958,157.616
C08860=1045.865,290.652,390.370,172.093,39.954,157.615
C08861=1045.857,290.358,390.407,172.089,39.952,157.614
C08862=1045.850,290.110,390.439,172.086,39.949,157.613
C08863=1045.844,289.862,390.471,172.083,39.946,157.613
C08864=1045.837,289.615,390.503,172.079,39.943,157.612
C08865=1045.831,289.367,390.534,172.076,39.941,157.611
C08866=1045.824,289.119,390.566,172.072,39.938,157.611
C08867=1045.818,288.871,390.598,172.070,39.935,157.610
C08868=1045.811,288.623,390.630,172.066,39.932,157.609
C08869=1045.804,288.375,390.661,172.062,39.930,157.608
C08870=1045.797,288.128,390.693,172.059,39.927,157.608
C08871=1045.791,287.880,390.725,172.056,39.924,157.607
C08872=1045.784,287.632,390.757,172.053,39.921,157.606
C08873=1045.778,287.384,390.788,172.049,39.919,157.605
C08874=1045.771,287.136,390.820,172.046,39.916,157.605
C08875=1045.764,286.889,390.852,172.043,39.913,157.604
C08876=1045.757,286.641,390.883,172.039,39.910,157.603
C08877=1045.750,286.393,390.915,172.036,39.908,157.603
C08878=1045.744,286.145,390.946,172.033,39.905,157.602
C08879=1045.737,285.897,390.978,172.030,39.903,157.601
C08880=1045.730,285.649,391.009,172.026,39.900,157.600
C08881=1045.724,285.401,391.040,172.023,39.897,157.600
C08882=1045.718,285.153,391.072,172.020,39.894,157.599
C08883=1045.711,284.905,391.104,172.017,39.892,157.598
C08884=1045.704,284.657,391.135,172.013,39.889,157.598
C08885=1045.697,284.410,391.167,172.010,39.887,157.597
C08886=1045.691,284.162,391.198,172.007,39.884,157.596
C08887=1045.684,283.914,391.230,172.003,39.881,157.595
C08888=1045.677,283.666,391.261,172.000,39.878,157.595
C08889=1045.671,283.418,391.292,171.997,39.876,157.594
C08890=1045.664,283.170,391.324,171.994,39.873,157.593
C08891=1045.657,282.922,391.355,171.990,39.871,157.593
C08892=1045.651,282.674,391.386,171.988,39.868,157.592
C08893=1045.644,282.426,391.418,171.984,39.865,157.591
C08894=1045.637,282.178,391.449,171.981,39.863,157.591
C08895=1045.630,281.930,391.480,171.977,39.860,157.590
C08896=1045.624,281.682,391.512,171.975,39.857,157.589
C08897=1045.618,281.435,391.543,171.971,39.855,157.588
C08898=1045.611,281.186,391.574,171.968,39.852,157.588
C08899=1045.605,280.938,391.605,171.965,39.850,157.587
C08900=1045.598,280.690,391.636,171.962,39.847,157.586
C08901=1045.591,280.443,391.668,171.959,39.844,157.586
C08902=1045.585,280.194,391.699,171.955,39.841,157.585
C08903=1045.579,279.947,391.730,171.953,39.839,157.584
C08904=1045.572,279.699,391.761,171.949,39.836,157.583
C08905=1045.565,279.451,391.793,171.946,39.834,157.583
C08906=1045.559,279.203,391.823,171.943,39.831,157.582
C08907=1045.552,278.955,391.855,171.940,39.828,157.581
C08908=1045.545,278.707,391.886,171.936,39.826,157.581
C08909=1045.539,278.459,391.916,171.934,39.823,157.580
C08910=1045.532,278.211,391.947,171.930,39.820,157.579
C08911=1045.525,277.963,391.978,171.927,39.818,157.579
C08912=1045.519,277.715,392.009,171.925,39.815,157.578
C08913=1045.512,277.467,392.040,171.921,39.813,157.577
C08914=1045.504,277.185,392.075,171.917,39.810,157.576
C08915=1045.497,276.903,392.110,171.914,39.807,157.576
C08916=1045.490,276.621,392.146,171.910,39.804,157.575
C08917=1045.482,276.338,392.181,171.907,39.801,157.574
C08918=1045.475,276.091,392.212,171.904,39.798,157.573
C08919=1045.469,275.842,392.242,171.900,39.796,157.573
C08920=1045.462,275.594,392.273,171.898,39.793,157.572
C08921=1045.455,275.346,392.304,171.894,39.790,157.571
C08922=1045.449,275.098,392.334,171.891,39.788,157.571
C08923=1045.443,274.851,392.366,171.889,39.785,157.570
C08924=1045.435,274.602,392.396,171.885,39.783,157.569
C08925=1045.429,274.354,392.427,171.882,39.780,157.569
C08926=1045.423,274.107,392.458,171.879,39.778,157.568
C08927=1045.416,273.858,392.488,171.876,39.775,157.567
C08928=1045.409,273.610,392.518,171.873,39.773,157.567
C08929=1045.403,273.362,392.550,171.870,39.770,157.566
C08930=1045.396,273.114,392.580,171.867,39.768,157.565
C08931=1045.390,272.866,392.610,171.864,39.765,157.565
C08932=1045.383,272.618,392.642,171.861,39.763,157.564
C08933=1045.376,272.371,392.672,171.858,39.760,157.563
C08934=1045.370,272.122,392.702,171.855,39.757,157.563
C08935=1045.363,271.873,392.733,171.852,39.755,157.562
C08936=1045.357,271.627,392.763,171.849,39.752,157.561
C08937=1045.350,271.378,392.794,171.845,39.750,157.561
C08938=1045.343,271.130,392.824,171.843,39.747,157.560
C08939=1045.337,270.882,392.855,171.840,39.745,157.559
C08940=1045.330,270.634,392.885,171.836,39.742,157.559
C08941=1045.324,270.385,392.916,171.834,39.739,157.558
C08942=1045.317,270.138,392.946,171.831,39.737,157.557
C08943=1045.310,269.890,392.977,171.827,39.734,157.557
C08944=1045.303,269.642,393.007,171.825,39.732,157.556
C08945=1045.297,269.394,393.037,171.822,39.729,157.555
C08946=1045.290,269.146,393.067,171.818,39.727,157.555
C08947=1045.284,268.897,393.098,171.816,39.724,157.554
C08948=1045.277,268.650,393.128,171.813,39.722,157.553
C08949=1045.271,268.401,393.158,171.809,39.719,157.553
C08950=1045.264,268.154,393.188,171.807,39.717,157.552
C08951=1045.258,267.905,393.219,171.804,39.714,157.551
C08952=1045.251,267.657,393.249,171.801,39.712,157.551
C08953=1045.245,267.409,393.279,171.798,39.709,157.550
C08954=1045.238,267.161,393.310,171.795,39.707,157.550
C08955=1045.231,266.913,393.339,171.792,39.704,157.549
C08956=1045.225,266.665,393.370,171.789,39.702,157.548
C08957=1045.218,266.417,393.400,171.786,39.699,157.548
C08958=1045.211,266.169,393.430,171.784,39.697,157.547
C08959=1045.205,265.920,393.460,171.780,39.694,157.546
C08960=1045.198,265.672,393.490,171.777,39.692,157.546
C08961=1045.191,265.424,393.520,171.775,39.689,157.545
C08962=1045.185,265.176,393.550,171.772,39.687,157.544
C08963=1045.178,264.928,393.580,171.768,39.684,157.544
C08964=1045.172,264.681,393.610,171.766,39.682,157.543
C08965=1045.166,264.431,393.640,171.763,39.679,157.542
C08966=1045.158,264.183,393.670,171.760,39.677,157.542
C08967=1045.152,263.936,393.700,171.757,39.674,157.541
C08968=1045.145,263.687,393.731,171.754,39.672,157.540
C08969=1045.139,263.439,393.760,171.751,39.669,157.540
C08970=1045.132,263.162,393.793,171.748,39.667,157.539
C08971=1045.124,262.884,393.827,171.745,39.664,157.538
C08972=1045.117,262.606,393.860,171.741,39.661,157.538
C08973=1045.110,262.328,393.894,171.739,39.658,157.537
C08974=1045.103,262.080,393.924,171.736,39.655,157.536
C08975=1045.097,261.832,393.953,171.732,39.653,157.536
C08976=1045.090,261.584,393.983,171.730,39.651,157.535
C08977=1045.083,261.335,394.012,171.727,39.649,157.535
C08978=1045.076,261.088,394.042,171.724,39.646,157.534
C08979=1045.069,260.839,394.072,171.721,39.644,157.533
C08980=1045.063,260.591,394.101,171.718,39.641,157.533
C08981=1045.056,260.343,394.131,171.716,39.639,157.532
C08982=1045.049,260.095,394.161,171.713,39.636,157.531
C08983=1045.042,259.847,394.191,171.709,39.634,157.531
C08984=1045.036,259.599,394.220,171.707,39.631,157.530
C08985=1045.028,259.351,394.249,171.704,39.629,157.529
C08986=1045.022,259.103,394.278,171.702,39.627,157.529
C08987=1045.016,258.854,394.307,171.699,39.625,157.528
C08988=1045.008,258.606,394.337,171.695,39.622,157.528
C08989=1045.002,258.358,394.366,171.693,39.620,157.527
C08990=1044.995,258.110,394.397,171.690,39.617,157.526
C08991=1044.989,257.862,394.426,171.688,39.614,157.526
C08992=1044.982,257.613,394.455,171.685,39.612,157.525
C08993=1044.975,257.365,394.485,171.681,39.610,157.525
C08994=1044.969,257.117,394.514,171.679,39.607,157.524
C08995=1044.962,256.868,394.543,171.676,39.605,157.523
C08996=1044.956,256.621,394.573,171.674,39.603,157.523
C08997=1044.949,256.372,394.602,171.671,39.600,157.522
C08998=1044.943,256.124,394.631,171.667,39.598,157.521
C08999=1044.935,255.876,394.662,171.665,39.595,157.521
C09000=1044.929,255.628,394.691,171.662,39.593,157.520
C09001=1044.922,255.380,394.719,171.659,39.590,157.520
C09002=1044.915,255.132,394.749,171.657,39.588,157.519
C09003=1044.909,254.883,394.778,171.654,39.586,157.518
C09004=1044.903,254.635,394.807,171.652,39.583,157.518
C09005=1044.896,254.386,394.837,171.648,39.581,157.517
C09006=1044.889,254.139,394.866,171.645,39.578,157.517
C09007=1044.883,253.891,394.895,171.643,39.576,157.516
C09008=1044.876,253.642,394.925,171.640,39.573,157.515
C09009=1044.870,253.394,394.954,171.638,39.571,157.515
C09010=1044.864,253.146,394.983,171.635,39.568,157.514
C09011=1044.857,252.897,395.012,171.632,39.566,157.513
C09012=1044.850,252.649,395.042,171.630,39.564,157.513
C09013=1044.843,252.402,395.071,171.626,39.561,157.512
C09014=1044.837,252.153,395.100,171.624,39.559,157.512
C09015=1044.830,251.905,395.129,171.621,39.556,157.511
C09016=1044.824,251.656,395.158,171.618,39.554,157.510
C09017=1044.818,251.408,395.187,171.616,39.551,157.510
C09018=1044.811,251.159,395.216,171.613,39.549,157.509
C09019=1044.805,250.911,395.246,171.610,39.546,157.508
C09020=1044.798,250.663,395.275,171.608,39.544,157.508
C09021=1044.792,250.415,395.304,171.605,39.542,157.507
C09022=1044.785,250.167,395.332,171.603,39.539,157.507
C09023=1044.778,249.918,395.361,171.600,39.537,157.506
C09024=1044.772,249.671,395.391,171.597,39.534,157.505
C09025=1044.765,249.423,395.420,171.594,39.531,157.505
C09026=1044.758,249.143,395.452,171.591,39.529,157.504
C09027=1044.752,248.864,395.485,171.589,39.526,157.503
C09028=1044.744,248.585,395.518,171.586,39.523,157.503
C09029=1044.737,248.306,395.550,171.582,39.521,157.502
C09030=1044.730,248.058,395.580,171.580,39.518,157.501
C09031=1044.724,247.809,395.609,171.577,39.516,157.501
C09032=1044.717,247.561,395.638,171.574,39.513,157.500
C09033=1044.710,247.313,395.666,171.572,39.511,157.500
C09034=1044.704,247.065,395.695,171.569,39.508,157.499
C09035=1044.698,246.816,395.724,171.567,39.506,157.498
C09036=1044.692,246.568,395.753,171.564,39.503,157.498
C09037=1044.686,246.320,395.782,171.561,39.501,157.497
C09038=1044.679,246.071,395.811,171.559,39.498,157.496
C09039=1044.673,245.823,395.840,171.556,39.496,157.496
C09040=1044.666,245.575,395.869,171.553,39.493,157.495
C09041=1044.659,245.327,395.898,171.551,39.491,157.495
C09042=1044.653,245.078,395.926,171.548,39.489,157.494
C09043=1044.646,244.830,395.955,171.546,39.486,157.493
C09044=1044.640,244.582,395.984,171.543,39.484,157.493
C09045=1044.634,244.333,396.012,171.541,39.481,157.492
C09046=1044.627,244.085,396.041,171.538,39.479,157.491
C09047=1044.620,243.837,396.070,171.535,39.476,157.491
C09048=1044.613,243.589,396.098,171.533,39.474,157.490
C09049=1044.607,243.340,396.127,171.530,39.472,157.490
C09050=1044.601,243.092,396.156,171.527,39.469,157.489
C09051=1044.594,242.844,396.184,171.525,39.467,157.488
C09052=1044.588,242.595,396.212,171.522,39.464,157.488
C09053=1044.581,242.348,396.241,171.520,39.462,157.487
C09054=1044.575,242.099,396.269,171.517,39.459,157.487
C09055=1044.569,241.850,396.299,171.515,39.457,157.486
C09056=1044.562,241.602,396.327,171.512,39.455,157.486
C09057=1044.556,241.353,396.355,171.509,39.452,157.485
C09058=1044.549,241.106,396.384,171.507,39.449,157.484
C09059=1044.542,240.857,396.411,171.504,39.447,157.484
C09060=1044.536,240.609,396.441,171.502,39.445,157.483
C09061=1044.529,240.361,396.468,171.499,39.443,157.483
C09062=1044.523,240.112,396.497,171.497,39.440,157.482
C09063=1044.516,239.864,396.525,171.494,39.437,157.481
C09064=1044.509,239.616,396.553,171.491,39.435,157.481
C09065=1044.503,239.367,396.582,171.490,39.433,157.480
C09066=1044.496,239.119,396.610,171.487,39.431,157.480
C09067=1044.489,238.871,396.638,171.485,39.428,157.479
C09068=1044.483,238.622,396.667,171.482,39.426,157.478
C09069=1044.476,238.374,396.695,171.479,39.423,157.478
C09070=1044.469,238.125,396.723,171.477,39.421,157.477
C09071=1044.463,237.877,396.751,171.474,39.419,157.477
C09072=1044.456,237.629,396.780,171.472,39.416,157.476
C09073=1044.450,237.380,396.807,171.469,39.414,157.475
C09074=1044.444,237.132,396.836,171.467,39.411,157.475
C09075=1044.437,236.884,396.864,171.464,39.409,157.474
C09076=1044.430,236.635,396.892,171.462,39.407,157.474
C09077=1044.423,236.387,396.920,171.459,39.404,157.473
C09078=1044.417,236.139,396.949,171.456,39.402,157.473
C09079=1044.410,235.890,396.976,171.454,39.400,157.472
C09080=1044.404,235.642,397.004,171.452,39.397,157.471
C09081=1044.398,235.393,397.032,171.450,39.394,157.471
C09082=1044.390,235.109,397.065,171.446,39.392,157.470
C09083=1044.383,234.823,397.097,171.443,39.389,157.469
C09084=1044.375,234.539,397.129,171.441,39.387,157.469
C09085=1044.368,234.254,397.161,171.438,39.384,157.468
C09086=1044.361,234.006,397.189,171.436,39.381,157.467
C09087=1044.354,233.757,397.217,171.433,39.378,157.467
C09088=1044.348,233.509,397.245,171.430,39.376,157.466
C09089=1044.342,233.260,397.273,171.428,39.374,157.466
C09090=1044.335,233.012,397.301,171.426,39.372,157.465
C09091=1044.328,232.763,397.328,171.424,39.369,157.465
C09092=1044.322,232.515,397.357,171.421,39.366,157.464
C09093=1044.315,232.267,397.385,171.418,39.364,157.463
C09094=1044.309,232.018,397.413,171.416,39.362,157.463
C09095=1044.302,231.770,397.441,171.413,39.360,157.462
C09096=1044.296,231.522,397.468,171.411,39.357,157.462
C09097=1044.290,231.273,397.496,171.409,39.354,157.461
C09098=1044.283,231.025,397.524,171.407,39.352,157.460
C09099=1044.277,230.776,397.552,171.404,39.350,157.460
C09100=1044.270,230.528,397.580,171.402,39.347,157.459
C09101=1044.263,230.280,397.607,171.399,39.345,157.459
C09102=1044.256,230.031,397.635,171.396,39.342,157.458
C09103=1044.250,229.783,397.663,171.395,39.340,157.457
C09104=1044.243,229.534,397.690,171.392,39.338,157.457
C09105=1044.237,229.287,397.718,171.390,39.335,157.456
C09106=1044.231,229.038,397.746,171.387,39.333,157.456
